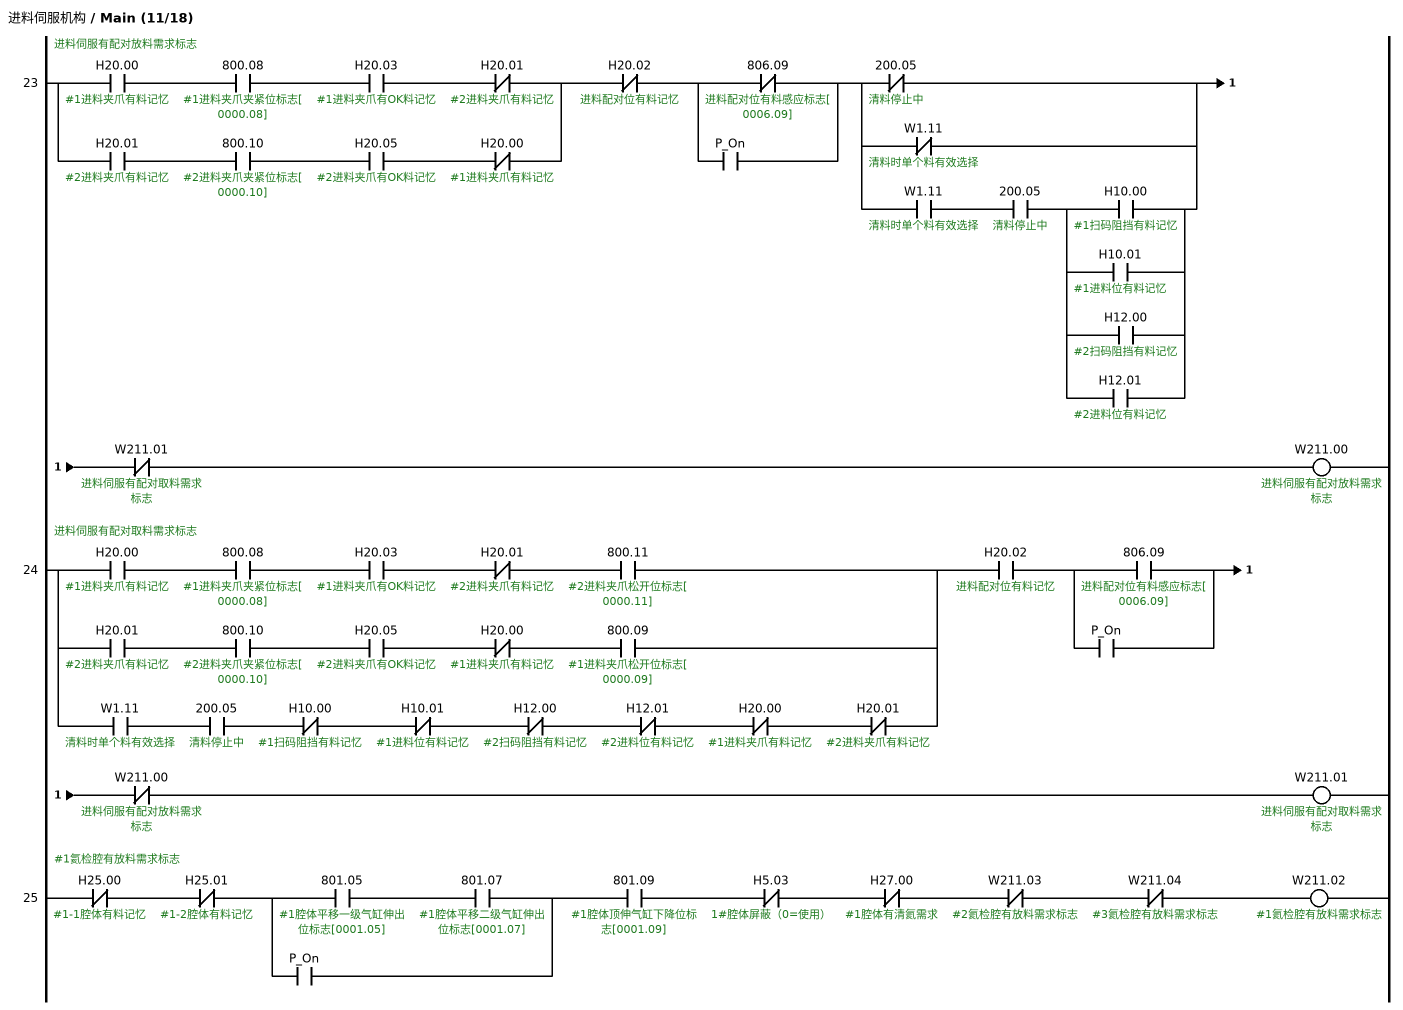
; [picture p72: 进料伺服机构 / Main, rungs 23-25]
; rung 23: 进料伺服有配对放料需求标志
LD H20.00  ; #1进料夹爪有料记忆
AND 800.08  ; #1进料夹爪夹紧位标志[0000.08]
AND H20.03  ; #1进料夹爪有OK料记忆
ANDNOT H20.01  ; #2进料夹爪有料记忆
LD H20.01  ; #2进料夹爪有料记忆
AND 800.10  ; #2进料夹爪夹紧位标志[0000.10]
AND H20.05  ; #2进料夹爪有OK料记忆
ANDNOT H20.00  ; #1进料夹爪有料记忆
ORLD
ANDNOT H20.02  ; 进料配对位有料记忆
LDNOT 806.09  ; 进料配对位有料感应标志[0006.09]
OR P_On
ANDLD
LDNOT 200.05  ; 清料停止中
ORNOT W1.11  ; 清料时单个料有效选择
LD W1.11  ; 清料时单个料有效选择
AND 200.05  ; 清料停止中
LD H10.00  ; #1扫码阻挡有料记忆
OR H10.01  ; #1进料位有料记忆
OR H12.00  ; #2扫码阻挡有料记忆
OR H12.01  ; #2进料位有料记忆
ANDLD
ORLD
ANDLD
ANDNOT W211.01  ; 进料伺服有配对取料需求标志
OUT W211.00  ; 进料伺服有配对放料需求标志
; rung 24: 进料伺服有配对取料需求标志
LD H20.00  ; #1进料夹爪有料记忆
AND 800.08  ; #1进料夹爪夹紧位标志[0000.08]
AND H20.03  ; #1进料夹爪有OK料记忆
ANDNOT H20.01  ; #2进料夹爪有料记忆
AND 800.11  ; #2进料夹爪松开位标志[0000.11]
LD H20.01  ; #2进料夹爪有料记忆
AND 800.10  ; #2进料夹爪夹紧位标志[0000.10]
AND H20.05  ; #2进料夹爪有OK料记忆
ANDNOT H20.00  ; #1进料夹爪有料记忆
AND 800.09  ; #1进料夹爪松开位标志[0000.09]
ORLD
LD W1.11  ; 清料时单个料有效选择
AND 200.05  ; 清料停止中
ANDNOT H10.00  ; #1扫码阻挡有料记忆
ANDNOT H10.01  ; #1进料位有料记忆
ANDNOT H12.00  ; #2扫码阻挡有料记忆
ANDNOT H12.01  ; #2进料位有料记忆
ANDNOT H20.00  ; #1进料夹爪有料记忆
ANDNOT H20.01  ; #2进料夹爪有料记忆
ORLD
AND H20.02  ; 进料配对位有料记忆
LD 806.09  ; 进料配对位有料感应标志[0006.09]
OR P_On
ANDLD
ANDNOT W211.00  ; 进料伺服有配对放料需求标志
OUT W211.01  ; 进料伺服有配对取料需求标志
; rung 25: #1氦检腔有放料需求标志
LDNOT H25.00  ; #1-1腔体有料记忆
ANDNOT H25.01  ; #1-2腔体有料记忆
LD 801.05  ; #1腔体平移一级气缸伸出位标志[0001.05]
AND 801.07  ; #1腔体平移二级气缸伸出位标志[0001.07]
OR P_On
ANDLD
AND 801.09  ; #1腔体顶伸气缸下降位标志[0001.09]
ANDNOT H5.03  ; 1#腔体屏蔽（0=使用）
ANDNOT H27.00  ; #1腔体有清氦需求
ANDNOT W211.03  ; #2氦检腔有放料需求标志
ANDNOT W211.04  ; #3氦检腔有放料需求标志
OUT W211.02  ; #1氦检腔有放料需求标志

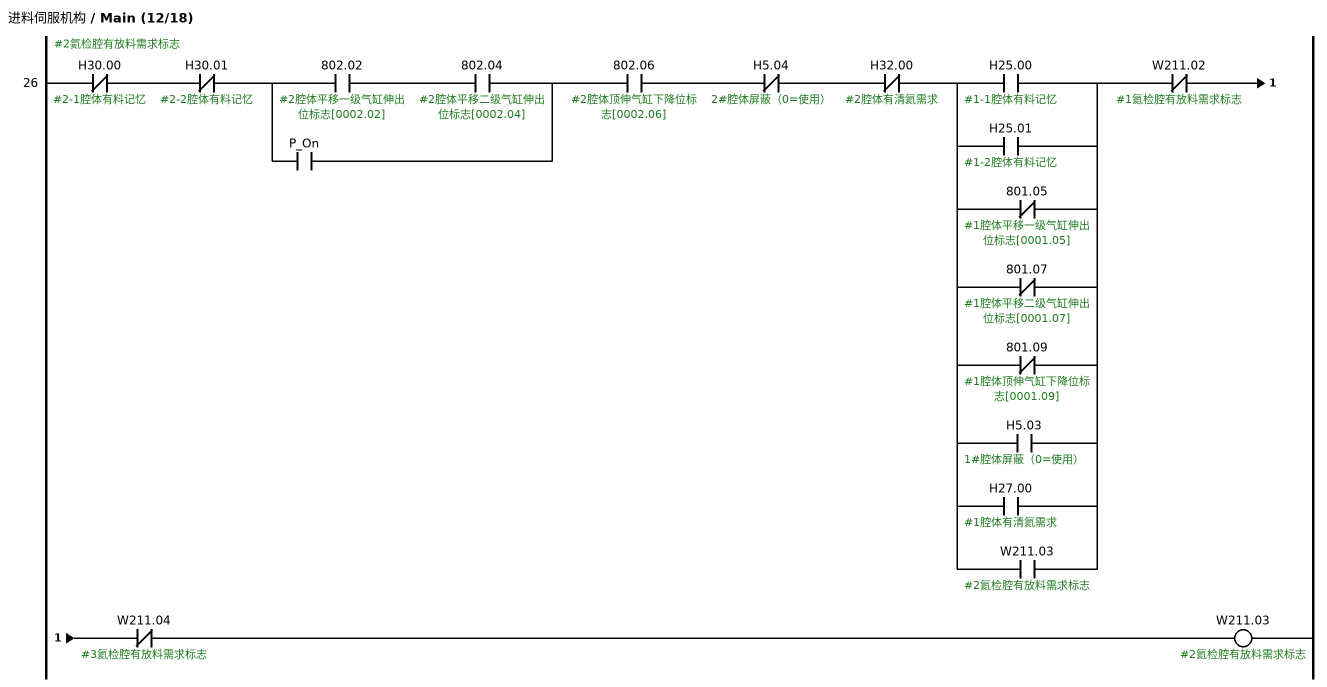
; rung 26: #2氦检腔有放料需求标志
LDNOT H30.00  ; #2-1腔体有料记忆
ANDNOT H30.01  ; #2-2腔体有料记忆
LD 802.02  ; #2腔体平移一级气缸伸出位标志[0002.02]
AND 802.04  ; #2腔体平移二级气缸伸出位标志[0002.04]
OR P_On
ANDLD
AND 802.06  ; #2腔体顶伸气缸下降位标志[0002.06]
ANDNOT H5.04  ; 2#腔体屏蔽（0=使用）
ANDNOT H32.00  ; #2腔体有清氦需求
LD H25.00  ; #1-1腔体有料记忆
OR H25.01  ; #1-2腔体有料记忆
ORNOT 801.05  ; #1腔体平移一级气缸伸出位标志[0001.05]
ORNOT 801.07  ; #1腔体平移二级气缸伸出位标志[0001.07]
ORNOT 801.09  ; #1腔体顶伸气缸下降位标志[0001.09]
OR H5.03  ; 1#腔体屏蔽（0=使用）
OR H27.00  ; #1腔体有清氦需求
OR W211.03  ; #2氦检腔有放料需求标志
ANDLD
ANDNOT W211.02  ; #1氦检腔有放料需求标志
ANDNOT W211.04  ; #3氦检腔有放料需求标志
OUT W211.03  ; #2氦检腔有放料需求标志

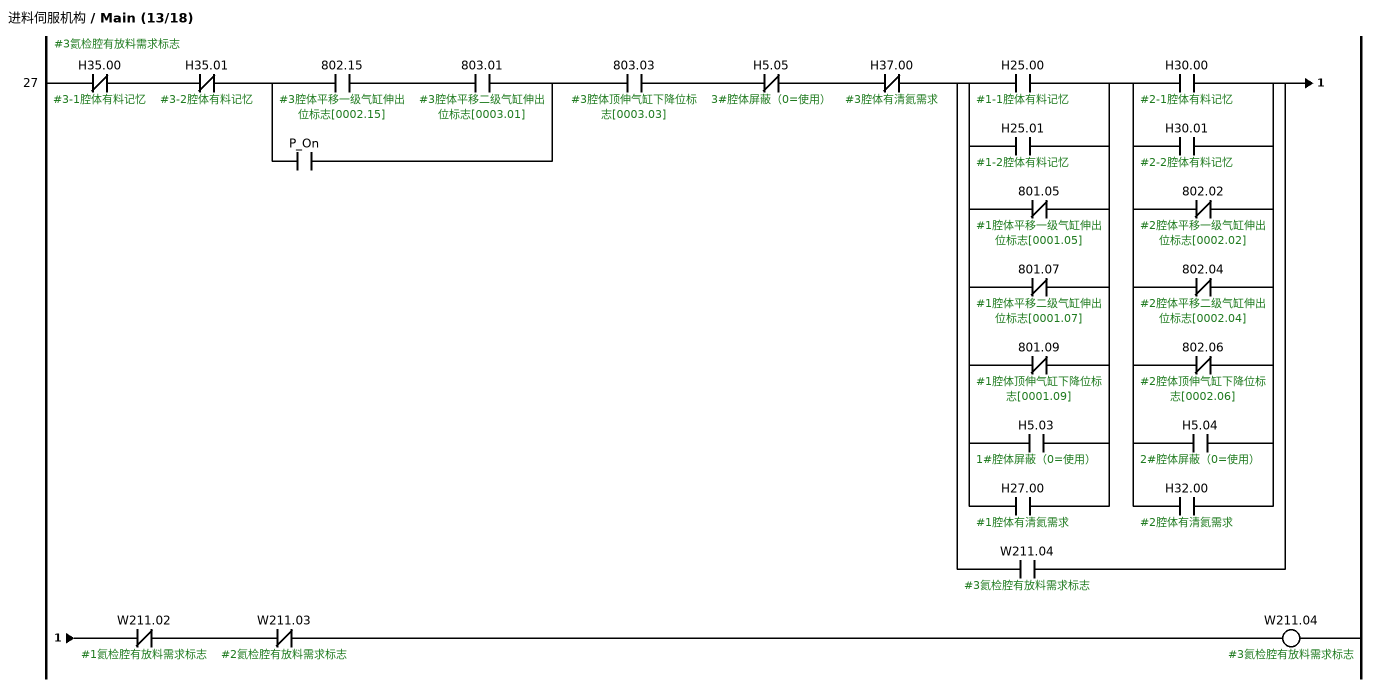
; rung 27: #3氦检腔有放料需求标志
LDNOT H35.00  ; #3-1腔体有料记忆
ANDNOT H35.01  ; #3-2腔体有料记忆
LD 802.15  ; #3腔体平移一级气缸伸出位标志[0002.15]
AND 803.01  ; #3腔体平移二级气缸伸出位标志[0003.01]
OR P_On
ANDLD
AND 803.03  ; #3腔体顶伸气缸下降位标志[0003.03]
ANDNOT H5.05  ; 3#腔体屏蔽（0=使用）
ANDNOT H37.00  ; #3腔体有清氦需求
LD H25.00  ; #1-1腔体有料记忆
OR H25.01  ; #1-2腔体有料记忆
ORNOT 801.05  ; #1腔体平移一级气缸伸出位标志[0001.05]
ORNOT 801.07  ; #1腔体平移二级气缸伸出位标志[0001.07]
ORNOT 801.09  ; #1腔体顶伸气缸下降位标志[0001.09]
OR H5.03  ; 1#腔体屏蔽（0=使用）
OR H27.00  ; #1腔体有清氦需求
LD H30.00  ; #2-1腔体有料记忆
OR H30.01  ; #2-2腔体有料记忆
ORNOT 802.02  ; #2腔体平移一级气缸伸出位标志[0002.02]
ORNOT 802.04  ; #2腔体平移二级气缸伸出位标志[0002.04]
ORNOT 802.06  ; #2腔体顶伸气缸下降位标志[0002.06]
OR H5.04  ; 2#腔体屏蔽（0=使用）
OR H32.00  ; #2腔体有清氦需求
ANDLD
OR W211.04  ; #3氦检腔有放料需求标志
ANDLD
ANDNOT W211.02  ; #1氦检腔有放料需求标志
ANDNOT W211.03  ; #2氦检腔有放料需求标志
OUT W211.04  ; #3氦检腔有放料需求标志

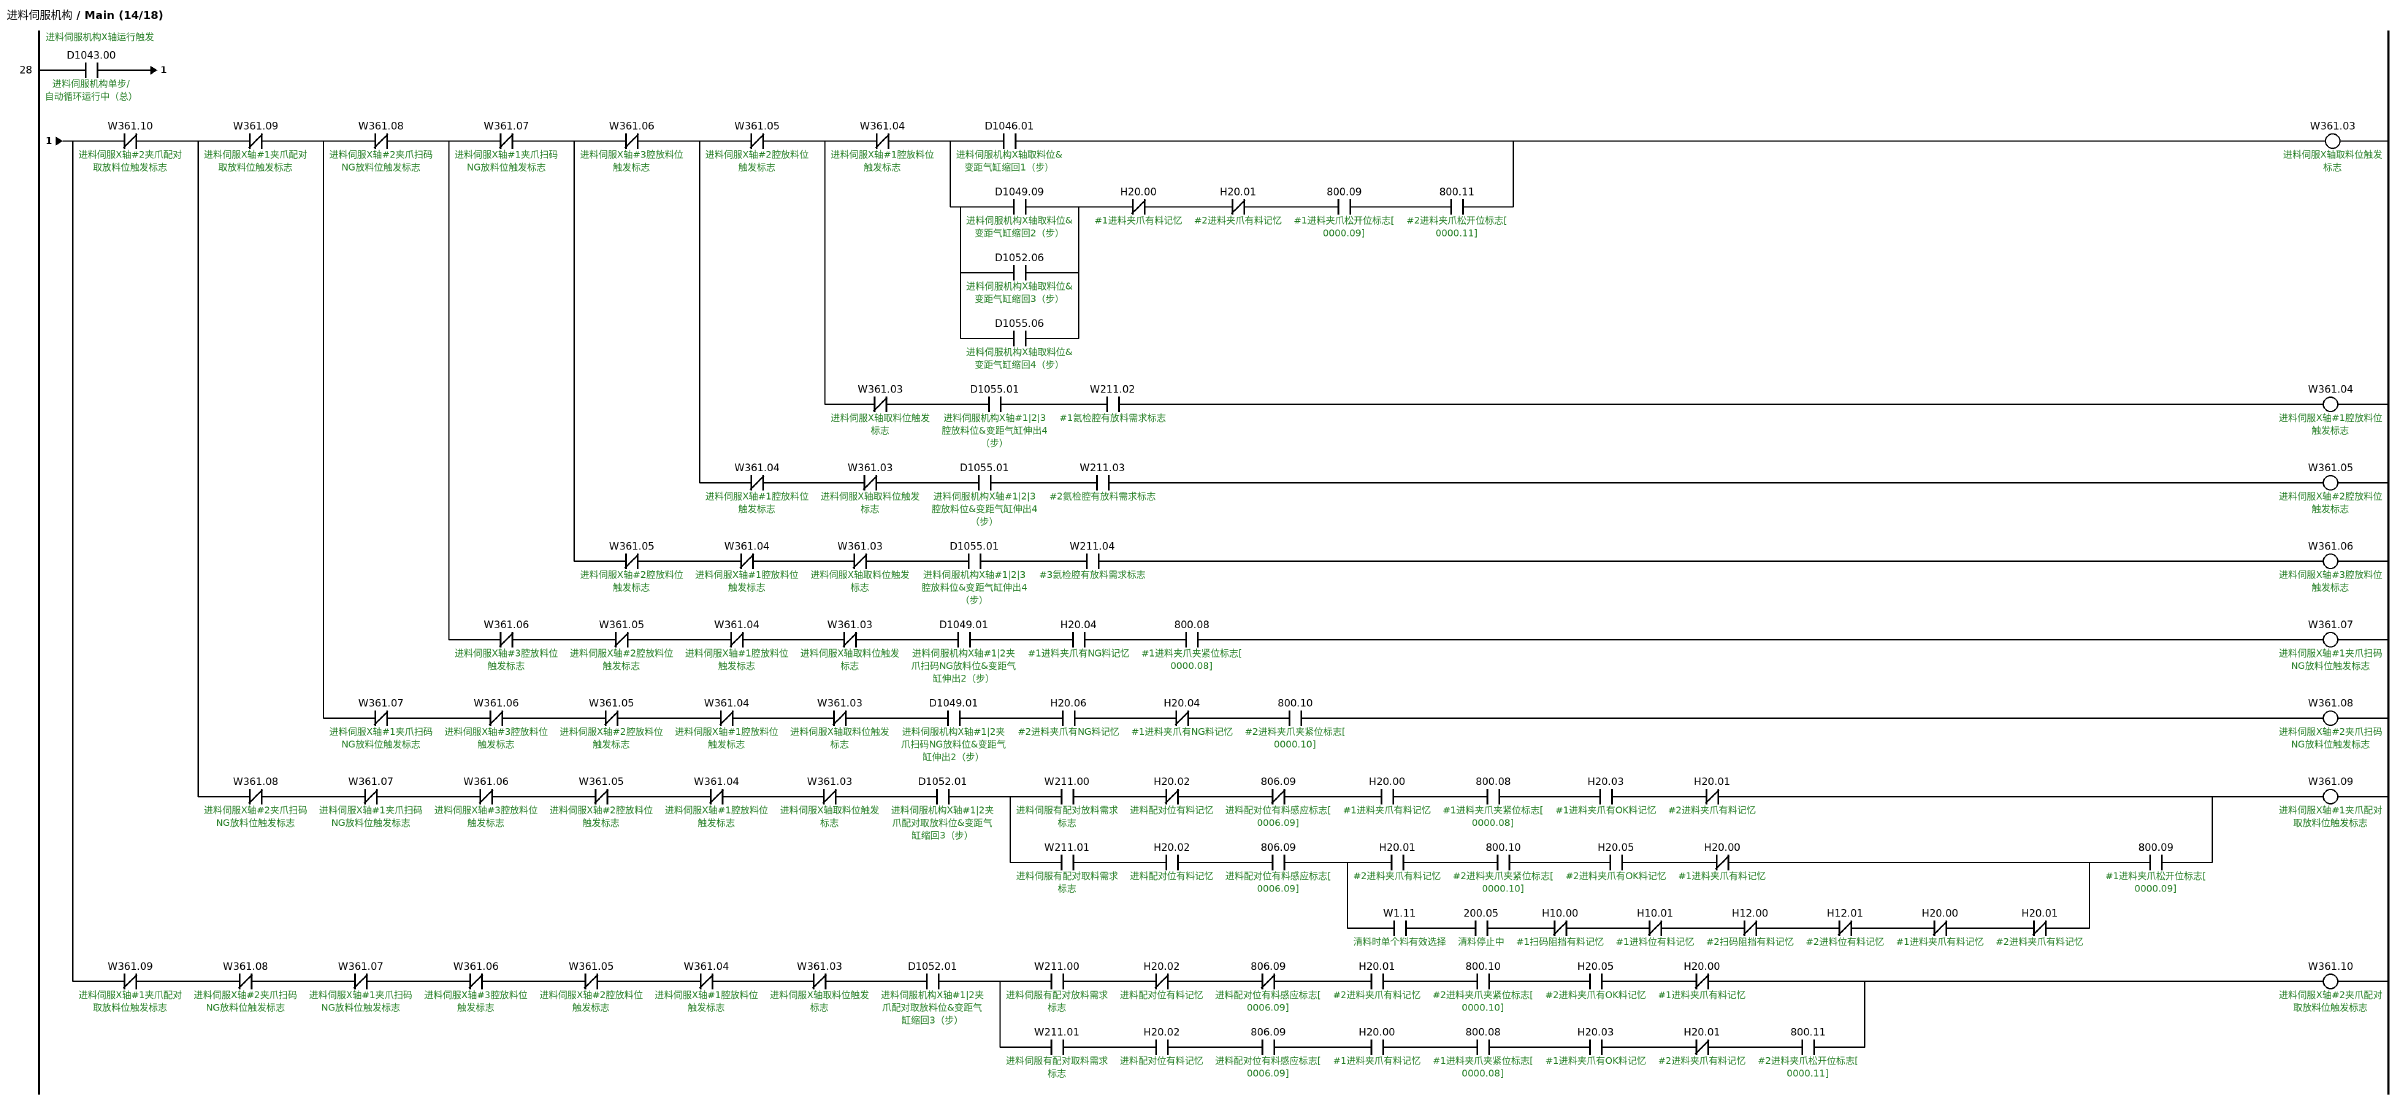
; rung 28: 进料伺服机构X轴运行触发
LD D1043.00  ; 进料伺服机构单步/自动循环运行中（总）
OUT TR0
ANDNOT W361.10  ; 进料伺服X轴#2夹爪配对取放料位触发标志
OUT TR1
ANDNOT W361.09  ; 进料伺服X轴#1夹爪配对取放料位触发标志
OUT TR2
ANDNOT W361.08  ; 进料伺服X轴#2夹爪扫码NG放料位触发标志
OUT TR3
ANDNOT W361.07  ; 进料伺服X轴#1夹爪扫码NG放料位触发标志
OUT TR4
ANDNOT W361.06  ; 进料伺服X轴#3腔放料位触发标志
OUT TR5
ANDNOT W361.05  ; 进料伺服X轴#2腔放料位触发标志
OUT TR6
ANDNOT W361.04  ; 进料伺服X轴#1腔放料位触发标志
LD D1046.01  ; 进料伺服机构X轴取料位&变距气缸缩回1（步）
LD D1049.09  ; 进料伺服机构X轴取料位&变距气缸缩回2（步）
OR D1052.06  ; 进料伺服机构X轴取料位&变距气缸缩回3（步）
OR D1055.06  ; 进料伺服机构X轴取料位&变距气缸缩回4（步）
ANDNOT H20.00  ; #1进料夹爪有料记忆
ANDNOT H20.01  ; #2进料夹爪有料记忆
AND 800.09  ; #1进料夹爪松开位标志[0000.09]
AND 800.11  ; #2进料夹爪松开位标志[0000.11]
ORLD
ANDLD
OUT W361.03  ; 进料伺服X轴取料位触发标志
LD TR6
ANDNOT W361.03  ; 进料伺服X轴取料位触发标志
AND D1055.01  ; 进料伺服机构X轴#1|2|3腔放料位&变距气缸伸出4（步）
AND W211.02  ; #1氦检腔有放料需求标志
OUT W361.04  ; 进料伺服X轴#1腔放料位触发标志
LD TR5
ANDNOT W361.04  ; 进料伺服X轴#1腔放料位触发标志
ANDNOT W361.03  ; 进料伺服X轴取料位触发标志
AND D1055.01  ; 进料伺服机构X轴#1|2|3腔放料位&变距气缸伸出4（步）
AND W211.03  ; #2氦检腔有放料需求标志
OUT W361.05  ; 进料伺服X轴#2腔放料位触发标志
LD TR4
ANDNOT W361.05  ; 进料伺服X轴#2腔放料位触发标志
ANDNOT W361.04  ; 进料伺服X轴#1腔放料位触发标志
ANDNOT W361.03  ; 进料伺服X轴取料位触发标志
AND D1055.01  ; 进料伺服机构X轴#1|2|3腔放料位&变距气缸伸出4（步）
AND W211.04  ; #3氦检腔有放料需求标志
OUT W361.06  ; 进料伺服X轴#3腔放料位触发标志
LD TR3
ANDNOT W361.06  ; 进料伺服X轴#3腔放料位触发标志
ANDNOT W361.05  ; 进料伺服X轴#2腔放料位触发标志
ANDNOT W361.04  ; 进料伺服X轴#1腔放料位触发标志
ANDNOT W361.03  ; 进料伺服X轴取料位触发标志
AND D1049.01  ; 进料伺服机构X轴#1|2夹爪扫码NG放料位&变距气缸伸出2（步）
AND H20.04  ; #1进料夹爪有NG料记忆
AND 800.08  ; #1进料夹爪夹紧位标志[0000.08]
OUT W361.07  ; 进料伺服X轴#1夹爪扫码NG放料位触发标志
LD TR2
ANDNOT W361.07  ; 进料伺服X轴#1夹爪扫码NG放料位触发标志
ANDNOT W361.06  ; 进料伺服X轴#3腔放料位触发标志
ANDNOT W361.05  ; 进料伺服X轴#2腔放料位触发标志
ANDNOT W361.04  ; 进料伺服X轴#1腔放料位触发标志
ANDNOT W361.03  ; 进料伺服X轴取料位触发标志
AND D1049.01  ; 进料伺服机构X轴#1|2夹爪扫码NG放料位&变距气缸伸出2（步）
AND H20.06  ; #2进料夹爪有NG料记忆
ANDNOT H20.04  ; #1进料夹爪有NG料记忆
AND 800.10  ; #2进料夹爪夹紧位标志[0000.10]
OUT W361.08  ; 进料伺服X轴#2夹爪扫码NG放料位触发标志
LD TR1
ANDNOT W361.08  ; 进料伺服X轴#2夹爪扫码NG放料位触发标志
ANDNOT W361.07  ; 进料伺服X轴#1夹爪扫码NG放料位触发标志
ANDNOT W361.06  ; 进料伺服X轴#3腔放料位触发标志
ANDNOT W361.05  ; 进料伺服X轴#2腔放料位触发标志
ANDNOT W361.04  ; 进料伺服X轴#1腔放料位触发标志
ANDNOT W361.03  ; 进料伺服X轴取料位触发标志
AND D1052.01  ; 进料伺服机构X轴#1|2夹爪配对取放料位&变距气缸缩回3（步）
LD W211.00  ; 进料伺服有配对放料需求标志
ANDNOT H20.02  ; 进料配对位有料记忆
ANDNOT 806.09  ; 进料配对位有料感应标志[0006.09]
AND H20.00  ; #1进料夹爪有料记忆
AND 800.08  ; #1进料夹爪夹紧位标志[0000.08]
AND H20.03  ; #1进料夹爪有OK料记忆
ANDNOT H20.01  ; #2进料夹爪有料记忆
LD W211.01  ; 进料伺服有配对取料需求标志
AND H20.02  ; 进料配对位有料记忆
AND 806.09  ; 进料配对位有料感应标志[0006.09]
LD H20.01  ; #2进料夹爪有料记忆
AND 800.10  ; #2进料夹爪夹紧位标志[0000.10]
AND H20.05  ; #2进料夹爪有OK料记忆
ANDNOT H20.00  ; #1进料夹爪有料记忆
LD W1.11  ; 清料时单个料有效选择
AND 200.05  ; 清料停止中
ANDNOT H10.00  ; #1扫码阻挡有料记忆
ANDNOT H10.01  ; #1进料位有料记忆
ANDNOT H12.00  ; #2扫码阻挡有料记忆
ANDNOT H12.01  ; #2进料位有料记忆
ANDNOT H20.00  ; #1进料夹爪有料记忆
ANDNOT H20.01  ; #2进料夹爪有料记忆
ORLD
ANDLD
AND 800.09  ; #1进料夹爪松开位标志[0000.09]
ORLD
ANDLD
OUT W361.09  ; 进料伺服X轴#1夹爪配对取放料位触发标志
LD TR0
ANDNOT W361.09  ; 进料伺服X轴#1夹爪配对取放料位触发标志
ANDNOT W361.08  ; 进料伺服X轴#2夹爪扫码NG放料位触发标志
ANDNOT W361.07  ; 进料伺服X轴#1夹爪扫码NG放料位触发标志
ANDNOT W361.06  ; 进料伺服X轴#3腔放料位触发标志
ANDNOT W361.05  ; 进料伺服X轴#2腔放料位触发标志
ANDNOT W361.04  ; 进料伺服X轴#1腔放料位触发标志
ANDNOT W361.03  ; 进料伺服X轴取料位触发标志
AND D1052.01  ; 进料伺服机构X轴#1|2夹爪配对取放料位&变距气缸缩回3（步）
LD W211.00  ; 进料伺服有配对放料需求标志
ANDNOT H20.02  ; 进料配对位有料记忆
ANDNOT 806.09  ; 进料配对位有料感应标志[0006.09]
AND H20.01  ; #2进料夹爪有料记忆
AND 800.10  ; #2进料夹爪夹紧位标志[0000.10]
AND H20.05  ; #2进料夹爪有OK料记忆
ANDNOT H20.00  ; #1进料夹爪有料记忆
LD W211.01  ; 进料伺服有配对取料需求标志
AND H20.02  ; 进料配对位有料记忆
AND 806.09  ; 进料配对位有料感应标志[0006.09]
AND H20.00  ; #1进料夹爪有料记忆
AND 800.08  ; #1进料夹爪夹紧位标志[0000.08]
AND H20.03  ; #1进料夹爪有OK料记忆
ANDNOT H20.01  ; #2进料夹爪有料记忆
AND 800.11  ; #2进料夹爪松开位标志[0000.11]
ORLD
ANDLD
OUT W361.10  ; 进料伺服X轴#2夹爪配对取放料位触发标志

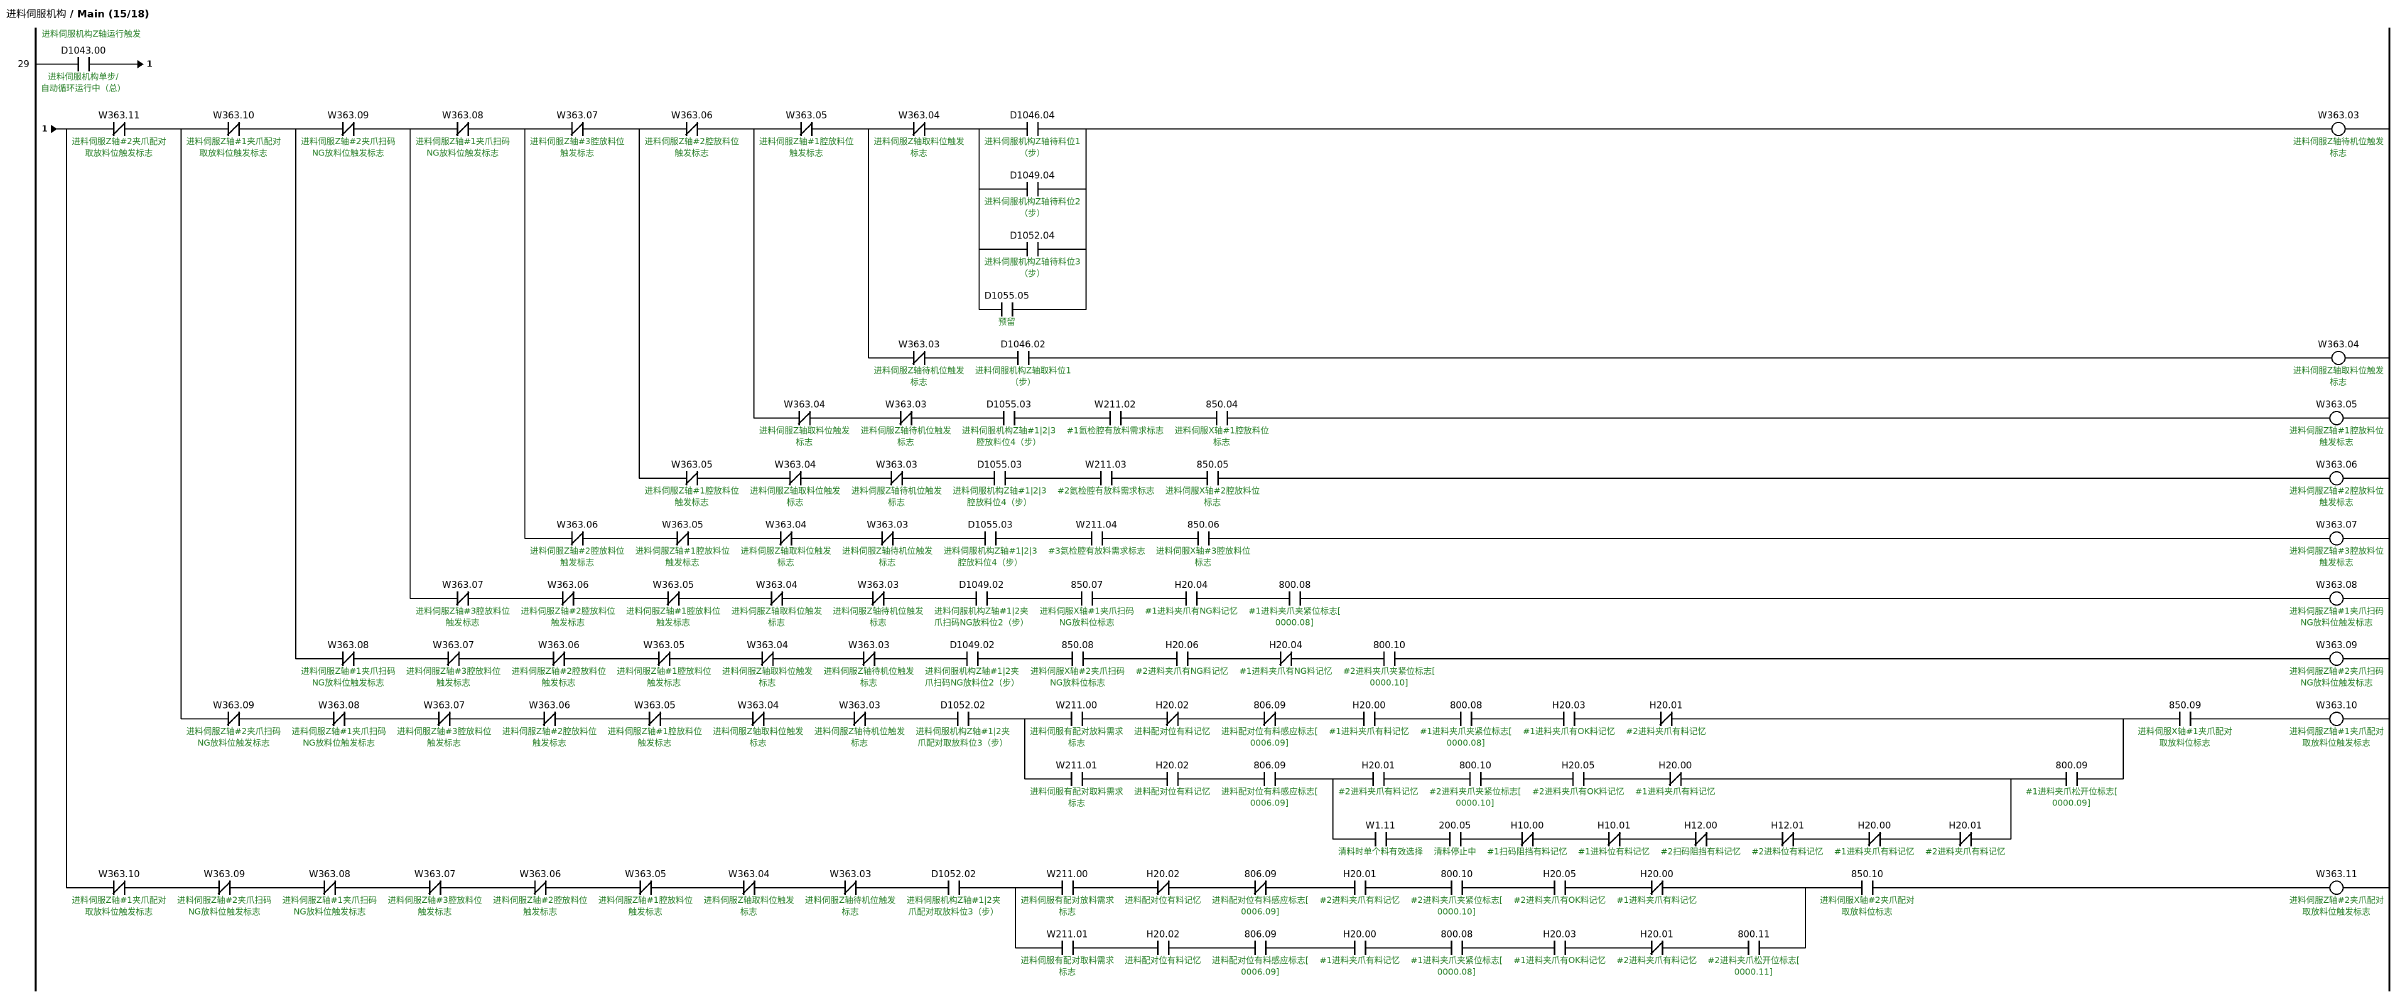
; rung 29: 进料伺服机构Z轴运行触发
LD D1043.00  ; 进料伺服机构单步/自动循环运行中（总）
OUT TR0
ANDNOT W363.11  ; 进料伺服Z轴#2夹爪配对取放料位触发标志
OUT TR1
ANDNOT W363.10  ; 进料伺服Z轴#1夹爪配对取放料位触发标志
OUT TR2
ANDNOT W363.09  ; 进料伺服Z轴#2夹爪扫码NG放料位触发标志
OUT TR3
ANDNOT W363.08  ; 进料伺服Z轴#1夹爪扫码NG放料位触发标志
OUT TR4
ANDNOT W363.07  ; 进料伺服Z轴#3腔放料位触发标志
OUT TR5
ANDNOT W363.06  ; 进料伺服Z轴#2腔放料位触发标志
OUT TR6
ANDNOT W363.05  ; 进料伺服Z轴#1腔放料位触发标志
OUT TR7
ANDNOT W363.04  ; 进料伺服Z轴取料位触发标志
LD D1046.04  ; 进料伺服机构Z轴待料位1（步）
OR D1049.04  ; 进料伺服机构Z轴待料位2（步）
OR D1052.04  ; 进料伺服机构Z轴待料位3（步）
OR D1055.05  ; 预留
ANDLD
OUT W363.03  ; 进料伺服Z轴待机位触发标志
LD TR7
ANDNOT W363.03  ; 进料伺服Z轴待机位触发标志
AND D1046.02  ; 进料伺服机构Z轴取料位1（步）
OUT W363.04  ; 进料伺服Z轴取料位触发标志
LD TR6
ANDNOT W363.04  ; 进料伺服Z轴取料位触发标志
ANDNOT W363.03  ; 进料伺服Z轴待机位触发标志
AND D1055.03  ; 进料伺服机构Z轴#1|2|3腔放料位4（步）
AND W211.02  ; #1氦检腔有放料需求标志
AND 850.04  ; 进料伺服X轴#1腔放料位标志
OUT W363.05  ; 进料伺服Z轴#1腔放料位触发标志
LD TR5
ANDNOT W363.05  ; 进料伺服Z轴#1腔放料位触发标志
ANDNOT W363.04  ; 进料伺服Z轴取料位触发标志
ANDNOT W363.03  ; 进料伺服Z轴待机位触发标志
AND D1055.03  ; 进料伺服机构Z轴#1|2|3腔放料位4（步）
AND W211.03  ; #2氦检腔有放料需求标志
AND 850.05  ; 进料伺服X轴#2腔放料位标志
OUT W363.06  ; 进料伺服Z轴#2腔放料位触发标志
LD TR4
ANDNOT W363.06  ; 进料伺服Z轴#2腔放料位触发标志
ANDNOT W363.05  ; 进料伺服Z轴#1腔放料位触发标志
ANDNOT W363.04  ; 进料伺服Z轴取料位触发标志
ANDNOT W363.03  ; 进料伺服Z轴待机位触发标志
AND D1055.03  ; 进料伺服机构Z轴#1|2|3腔放料位4（步）
AND W211.04  ; #3氦检腔有放料需求标志
AND 850.06  ; 进料伺服X轴#3腔放料位标志
OUT W363.07  ; 进料伺服Z轴#3腔放料位触发标志
LD TR3
ANDNOT W363.07  ; 进料伺服Z轴#3腔放料位触发标志
ANDNOT W363.06  ; 进料伺服Z轴#2腔放料位触发标志
ANDNOT W363.05  ; 进料伺服Z轴#1腔放料位触发标志
ANDNOT W363.04  ; 进料伺服Z轴取料位触发标志
ANDNOT W363.03  ; 进料伺服Z轴待机位触发标志
AND D1049.02  ; 进料伺服机构Z轴#1|2夹爪扫码NG放料位2（步）
AND 850.07  ; 进料伺服X轴#1夹爪扫码NG放料位标志
AND H20.04  ; #1进料夹爪有NG料记忆
AND 800.08  ; #1进料夹爪夹紧位标志[0000.08]
OUT W363.08  ; 进料伺服Z轴#1夹爪扫码NG放料位触发标志
LD TR2
ANDNOT W363.08  ; 进料伺服Z轴#1夹爪扫码NG放料位触发标志
ANDNOT W363.07  ; 进料伺服Z轴#3腔放料位触发标志
ANDNOT W363.06  ; 进料伺服Z轴#2腔放料位触发标志
ANDNOT W363.05  ; 进料伺服Z轴#1腔放料位触发标志
ANDNOT W363.04  ; 进料伺服Z轴取料位触发标志
ANDNOT W363.03  ; 进料伺服Z轴待机位触发标志
AND D1049.02  ; 进料伺服机构Z轴#1|2夹爪扫码NG放料位2（步）
AND 850.08  ; 进料伺服X轴#2夹爪扫码NG放料位标志
AND H20.06  ; #2进料夹爪有NG料记忆
ANDNOT H20.04  ; #1进料夹爪有NG料记忆
AND 800.10  ; #2进料夹爪夹紧位标志[0000.10]
OUT W363.09  ; 进料伺服Z轴#2夹爪扫码NG放料位触发标志
LD TR1
ANDNOT W363.09  ; 进料伺服Z轴#2夹爪扫码NG放料位触发标志
ANDNOT W363.08  ; 进料伺服Z轴#1夹爪扫码NG放料位触发标志
ANDNOT W363.07  ; 进料伺服Z轴#3腔放料位触发标志
ANDNOT W363.06  ; 进料伺服Z轴#2腔放料位触发标志
ANDNOT W363.05  ; 进料伺服Z轴#1腔放料位触发标志
ANDNOT W363.04  ; 进料伺服Z轴取料位触发标志
ANDNOT W363.03  ; 进料伺服Z轴待机位触发标志
AND D1052.02  ; 进料伺服机构Z轴#1|2夹爪配对取放料位3（步）
LD W211.00  ; 进料伺服有配对放料需求标志
ANDNOT H20.02  ; 进料配对位有料记忆
ANDNOT 806.09  ; 进料配对位有料感应标志[0006.09]
AND H20.00  ; #1进料夹爪有料记忆
AND 800.08  ; #1进料夹爪夹紧位标志[0000.08]
AND H20.03  ; #1进料夹爪有OK料记忆
ANDNOT H20.01  ; #2进料夹爪有料记忆
LD W211.01  ; 进料伺服有配对取料需求标志
AND H20.02  ; 进料配对位有料记忆
AND 806.09  ; 进料配对位有料感应标志[0006.09]
LD H20.01  ; #2进料夹爪有料记忆
AND 800.10  ; #2进料夹爪夹紧位标志[0000.10]
AND H20.05  ; #2进料夹爪有OK料记忆
ANDNOT H20.00  ; #1进料夹爪有料记忆
LD W1.11  ; 清料时单个料有效选择
AND 200.05  ; 清料停止中
ANDNOT H10.00  ; #1扫码阻挡有料记忆
ANDNOT H10.01  ; #1进料位有料记忆
ANDNOT H12.00  ; #2扫码阻挡有料记忆
ANDNOT H12.01  ; #2进料位有料记忆
ANDNOT H20.00  ; #1进料夹爪有料记忆
ANDNOT H20.01  ; #2进料夹爪有料记忆
ORLD
ANDLD
AND 800.09  ; #1进料夹爪松开位标志[0000.09]
ORLD
ANDLD
AND 850.09  ; 进料伺服X轴#1夹爪配对取放料位标志
OUT W363.10  ; 进料伺服Z轴#1夹爪配对取放料位触发标志
LD TR0
ANDNOT W363.10  ; 进料伺服Z轴#1夹爪配对取放料位触发标志
ANDNOT W363.09  ; 进料伺服Z轴#2夹爪扫码NG放料位触发标志
ANDNOT W363.08  ; 进料伺服Z轴#1夹爪扫码NG放料位触发标志
ANDNOT W363.07  ; 进料伺服Z轴#3腔放料位触发标志
ANDNOT W363.06  ; 进料伺服Z轴#2腔放料位触发标志
ANDNOT W363.05  ; 进料伺服Z轴#1腔放料位触发标志
ANDNOT W363.04  ; 进料伺服Z轴取料位触发标志
ANDNOT W363.03  ; 进料伺服Z轴待机位触发标志
AND D1052.02  ; 进料伺服机构Z轴#1|2夹爪配对取放料位3（步）
LD W211.00  ; 进料伺服有配对放料需求标志
ANDNOT H20.02  ; 进料配对位有料记忆
ANDNOT 806.09  ; 进料配对位有料感应标志[0006.09]
AND H20.01  ; #2进料夹爪有料记忆
AND 800.10  ; #2进料夹爪夹紧位标志[0000.10]
AND H20.05  ; #2进料夹爪有OK料记忆
ANDNOT H20.00  ; #1进料夹爪有料记忆
LD W211.01  ; 进料伺服有配对取料需求标志
AND H20.02  ; 进料配对位有料记忆
AND 806.09  ; 进料配对位有料感应标志[0006.09]
AND H20.00  ; #1进料夹爪有料记忆
AND 800.08  ; #1进料夹爪夹紧位标志[0000.08]
AND H20.03  ; #1进料夹爪有OK料记忆
ANDNOT H20.01  ; #2进料夹爪有料记忆
AND 800.11  ; #2进料夹爪松开位标志[0000.11]
ORLD
ANDLD
AND 850.10  ; 进料伺服X轴#2夹爪配对取放料位标志
OUT W363.11  ; 进料伺服Z轴#2夹爪配对取放料位触发标志

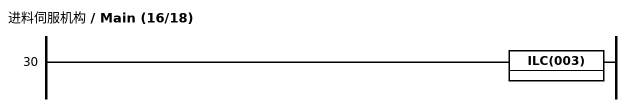
; rung 30
ILC(003)

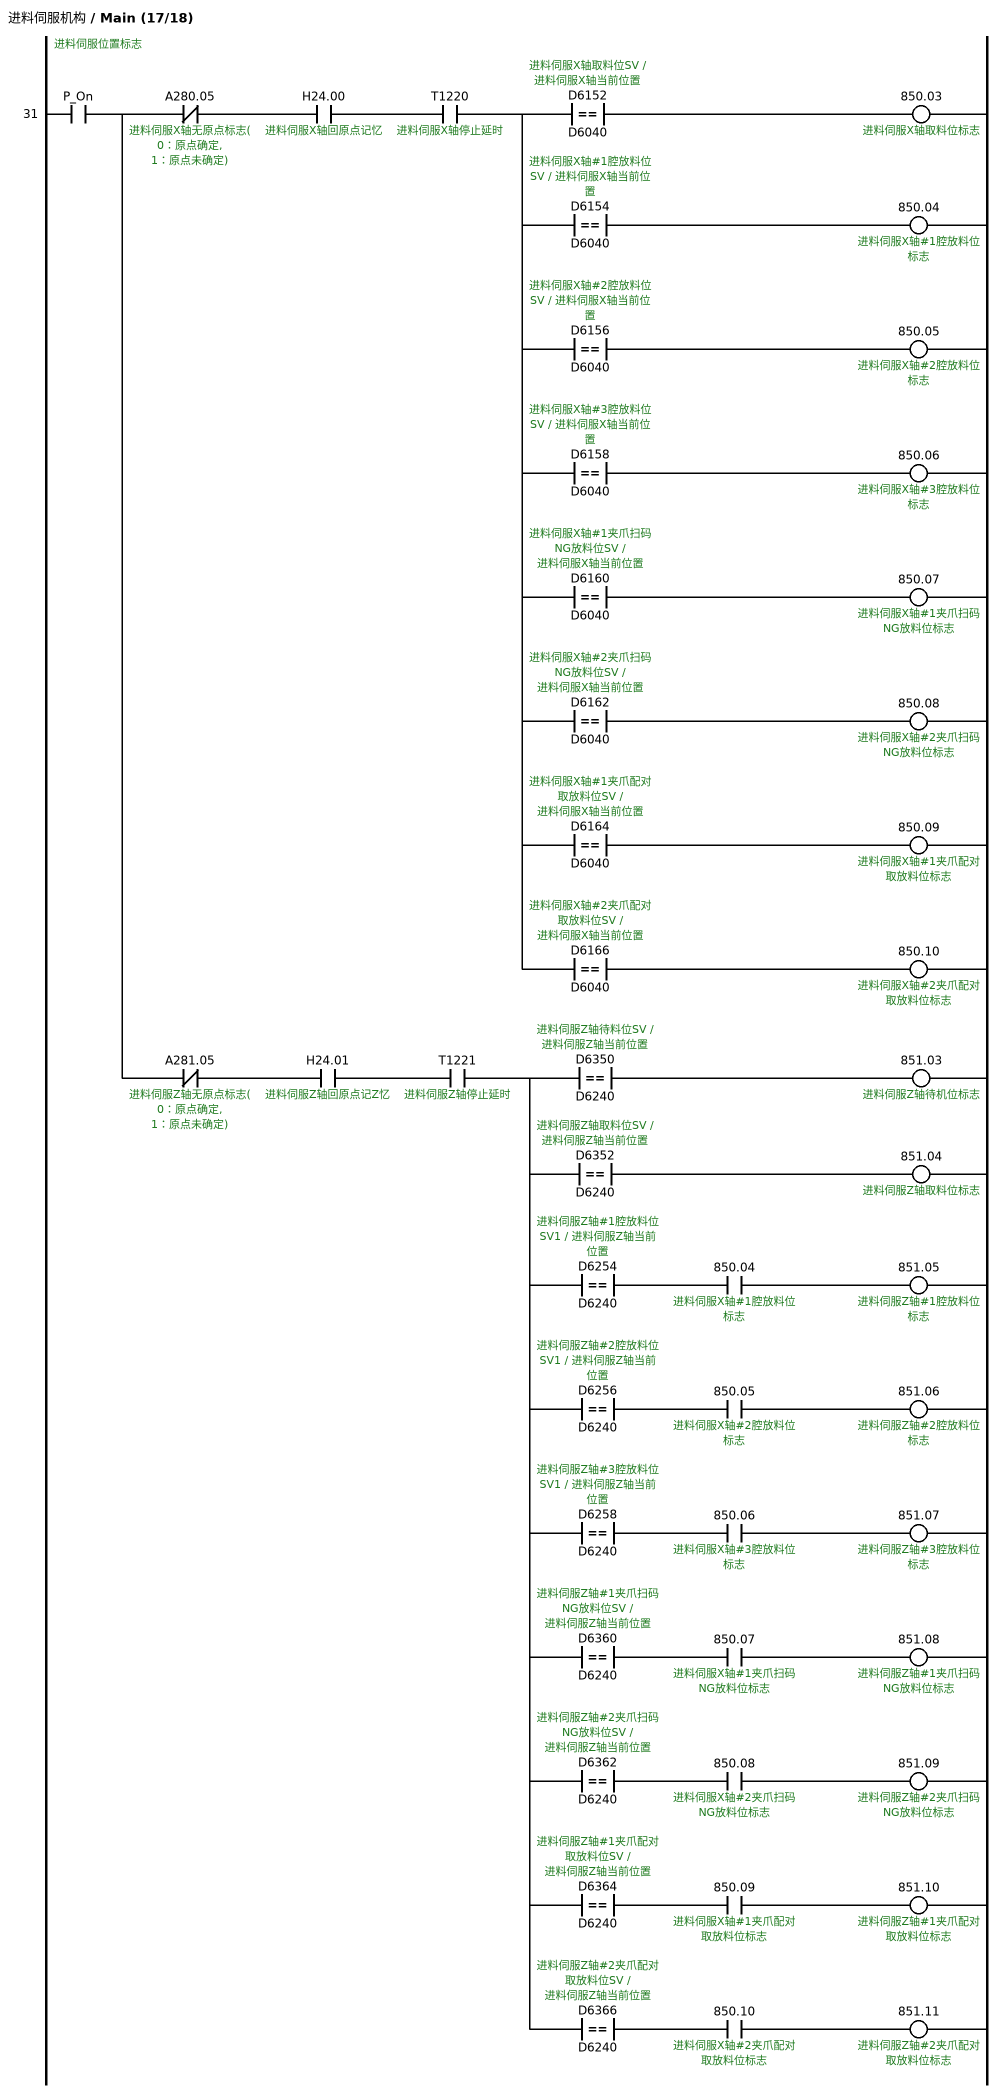
; rung 31: 进料伺服位置标志
LD P_On
OUT TR0
ANDNOT A280.05  ; 进料伺服X轴无原点标志(0：原点确定,1：原点未确定)
AND H24.00  ; 进料伺服X轴回原点记忆
AND T1220  ; 进料伺服X轴停止延时
OUT TR1
AND=SL(303) D6152 D6040  ; 进料伺服X轴取料位SV, 进料伺服X轴当前位置
OUT 850.03  ; 进料伺服X轴取料位标志
LD TR1
AND=SL(303) D6154 D6040  ; 进料伺服X轴#1腔放料位SV, 进料伺服X轴当前位置
OUT 850.04  ; 进料伺服X轴#1腔放料位标志
LD TR1
AND=SL(303) D6156 D6040  ; 进料伺服X轴#2腔放料位SV, 进料伺服X轴当前位置
OUT 850.05  ; 进料伺服X轴#2腔放料位标志
LD TR1
AND=SL(303) D6158 D6040  ; 进料伺服X轴#3腔放料位SV, 进料伺服X轴当前位置
OUT 850.06  ; 进料伺服X轴#3腔放料位标志
LD TR1
AND=SL(303) D6160 D6040  ; 进料伺服X轴#1夹爪扫码NG放料位SV, 进料伺服X轴当前位置
OUT 850.07  ; 进料伺服X轴#1夹爪扫码NG放料位标志
LD TR1
AND=SL(303) D6162 D6040  ; 进料伺服X轴#2夹爪扫码NG放料位SV, 进料伺服X轴当前位置
OUT 850.08  ; 进料伺服X轴#2夹爪扫码NG放料位标志
LD TR1
AND=SL(303) D6164 D6040  ; 进料伺服X轴#1夹爪配对取放料位SV, 进料伺服X轴当前位置
OUT 850.09  ; 进料伺服X轴#1夹爪配对取放料位标志
LD TR1
AND=SL(303) D6166 D6040  ; 进料伺服X轴#2夹爪配对取放料位SV, 进料伺服X轴当前位置
OUT 850.10  ; 进料伺服X轴#2夹爪配对取放料位标志
LD TR0
ANDNOT A281.05  ; 进料伺服Z轴无原点标志(0：原点确定,1：原点未确定)
AND H24.01  ; 进料伺服Z轴回原点记Z忆
AND T1221  ; 进料伺服Z轴停止延时
OUT TR0
AND=SL(303) D6350 D6240  ; 进料伺服Z轴待料位SV, 进料伺服Z轴当前位置
OUT 851.03  ; 进料伺服Z轴待机位标志
LD TR0
AND=SL(303) D6352 D6240  ; 进料伺服Z轴取料位SV, 进料伺服Z轴当前位置
OUT 851.04  ; 进料伺服Z轴取料位标志
LD TR0
AND=SL(303) D6254 D6240  ; 进料伺服Z轴#1腔放料位SV1, 进料伺服Z轴当前位置
AND 850.04  ; 进料伺服X轴#1腔放料位标志
OUT 851.05  ; 进料伺服Z轴#1腔放料位标志
LD TR0
AND=SL(303) D6256 D6240  ; 进料伺服Z轴#2腔放料位SV1, 进料伺服Z轴当前位置
AND 850.05  ; 进料伺服X轴#2腔放料位标志
OUT 851.06  ; 进料伺服Z轴#2腔放料位标志
LD TR0
AND=SL(303) D6258 D6240  ; 进料伺服Z轴#3腔放料位SV1, 进料伺服Z轴当前位置
AND 850.06  ; 进料伺服X轴#3腔放料位标志
OUT 851.07  ; 进料伺服Z轴#3腔放料位标志
LD TR0
AND=SL(303) D6360 D6240  ; 进料伺服Z轴#1夹爪扫码NG放料位SV, 进料伺服Z轴当前位置
AND 850.07  ; 进料伺服X轴#1夹爪扫码NG放料位标志
OUT 851.08  ; 进料伺服Z轴#1夹爪扫码NG放料位标志
LD TR0
AND=SL(303) D6362 D6240  ; 进料伺服Z轴#2夹爪扫码NG放料位SV, 进料伺服Z轴当前位置
AND 850.08  ; 进料伺服X轴#2夹爪扫码NG放料位标志
OUT 851.09  ; 进料伺服Z轴#2夹爪扫码NG放料位标志
LD TR0
AND=SL(303) D6364 D6240  ; 进料伺服Z轴#1夹爪配对取放料位SV, 进料伺服Z轴当前位置
AND 850.09  ; 进料伺服X轴#1夹爪配对取放料位标志
OUT 851.10  ; 进料伺服Z轴#1夹爪配对取放料位标志
LD TR0
AND=SL(303) D6366 D6240  ; 进料伺服Z轴#2夹爪配对取放料位SV, 进料伺服Z轴当前位置
AND 850.10  ; 进料伺服X轴#2夹爪配对取放料位标志
OUT 851.11  ; 进料伺服Z轴#2夹爪配对取放料位标志

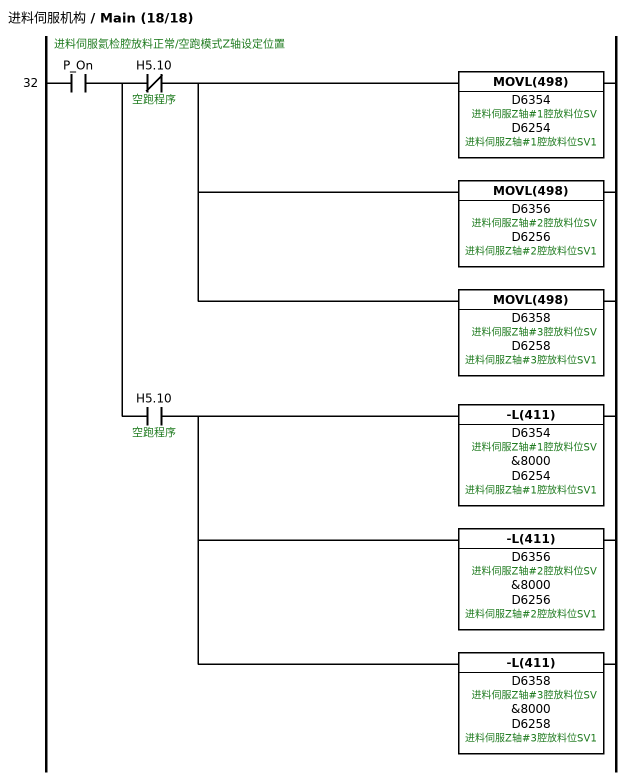
; rung 32: 进料伺服氦检腔放料正常/空跑模式Z轴设定位置
LD P_On
OUT TR0
ANDNOT H5.10  ; 空跑程序
MOVL(498) D6354 D6254  ; 进料伺服Z轴#1腔放料位SV, 进料伺服Z轴#1腔放料位SV1
MOVL(498) D6356 D6256  ; 进料伺服Z轴#2腔放料位SV, 进料伺服Z轴#2腔放料位SV1
MOVL(498) D6358 D6258  ; 进料伺服Z轴#3腔放料位SV, 进料伺服Z轴#3腔放料位SV1
LD TR0
AND H5.10  ; 空跑程序
-L(411) D6354 &8000 D6254  ; 进料伺服Z轴#1腔放料位SV, 进料伺服Z轴#1腔放料位SV1
-L(411) D6356 &8000 D6256  ; 进料伺服Z轴#2腔放料位SV, 进料伺服Z轴#2腔放料位SV1
-L(411) D6358 &8000 D6258  ; 进料伺服Z轴#3腔放料位SV, 进料伺服Z轴#3腔放料位SV1

### Section 进料伺服手动

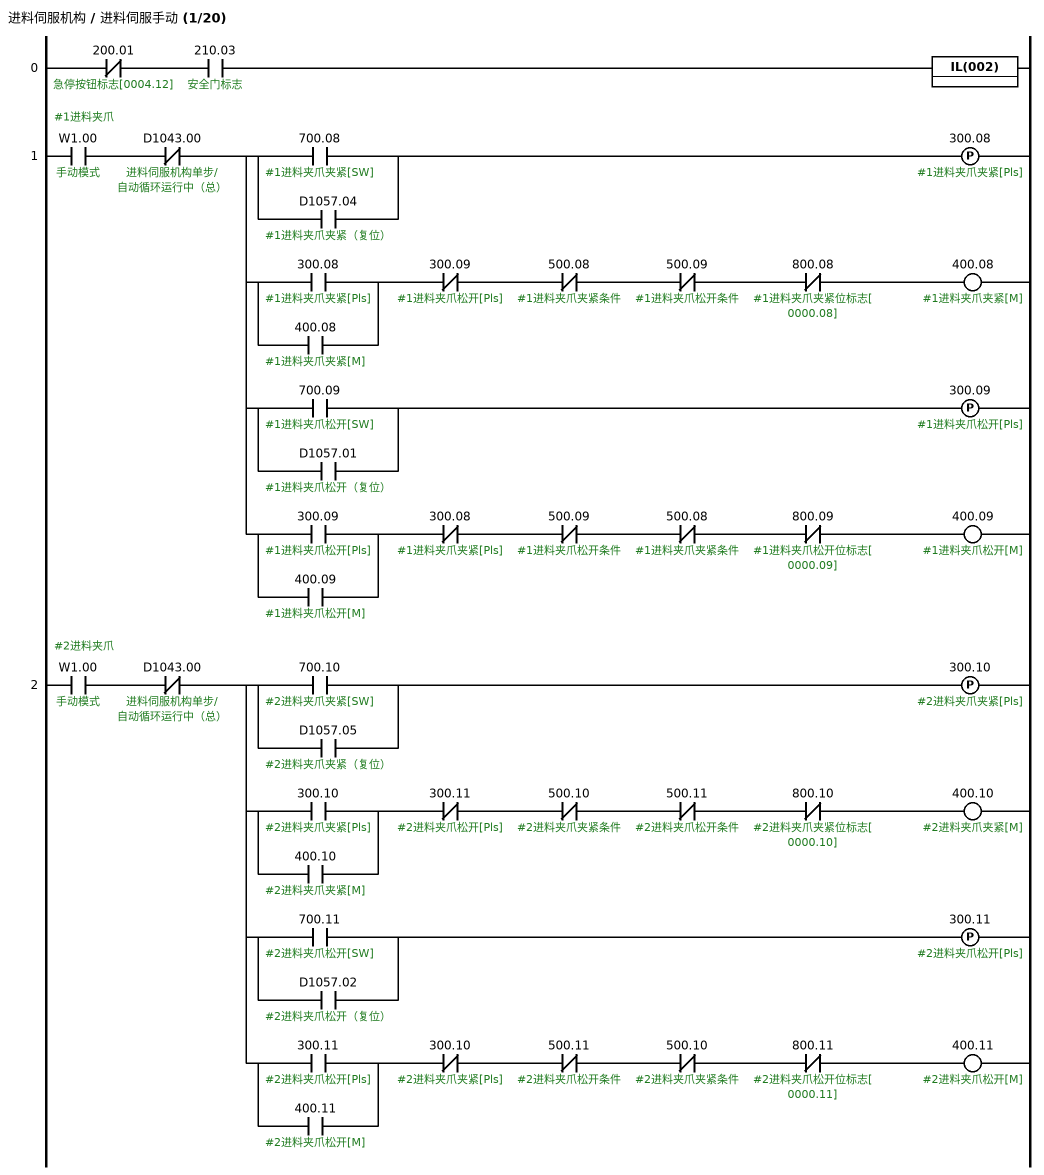
; rung 0
LDNOT 200.01  ; 急停按钮标志[0004.12]
AND 210.03  ; 安全门标志
IL(002)
; rung 1: #1进料夹爪
LD W1.00  ; 手动模式
ANDNOT D1043.00  ; 进料伺服机构单步/自动循环运行中（总）
OUT TR0
LD 700.08  ; #1进料夹爪夹紧[SW]
OR D1057.04  ; #1进料夹爪夹紧（复位）
ANDLD
DIFU(013) 300.08  ; #1进料夹爪夹紧[Pls]
LD TR0
LD 300.08  ; #1进料夹爪夹紧[Pls]
OR 400.08  ; #1进料夹爪夹紧[M]
ANDLD
ANDNOT 300.09  ; #1进料夹爪松开[Pls]
ANDNOT 500.08  ; #1进料夹爪夹紧条件
ANDNOT 500.09  ; #1进料夹爪松开条件
ANDNOT 800.08  ; #1进料夹爪夹紧位标志[0000.08]
OUT 400.08  ; #1进料夹爪夹紧[M]
LD TR0
LD 700.09  ; #1进料夹爪松开[SW]
OR D1057.01  ; #1进料夹爪松开（复位）
ANDLD
DIFU(013) 300.09  ; #1进料夹爪松开[Pls]
LD TR0
LD 300.09  ; #1进料夹爪松开[Pls]
OR 400.09  ; #1进料夹爪松开[M]
ANDLD
ANDNOT 300.08  ; #1进料夹爪夹紧[Pls]
ANDNOT 500.09  ; #1进料夹爪松开条件
ANDNOT 500.08  ; #1进料夹爪夹紧条件
ANDNOT 800.09  ; #1进料夹爪松开位标志[0000.09]
OUT 400.09  ; #1进料夹爪松开[M]
; rung 2: #2进料夹爪
LD W1.00  ; 手动模式
ANDNOT D1043.00  ; 进料伺服机构单步/自动循环运行中（总）
OUT TR0
LD 700.10  ; #2进料夹爪夹紧[SW]
OR D1057.05  ; #2进料夹爪夹紧（复位）
ANDLD
DIFU(013) 300.10  ; #2进料夹爪夹紧[Pls]
LD TR0
LD 300.10  ; #2进料夹爪夹紧[Pls]
OR 400.10  ; #2进料夹爪夹紧[M]
ANDLD
ANDNOT 300.11  ; #2进料夹爪松开[Pls]
ANDNOT 500.10  ; #2进料夹爪夹紧条件
ANDNOT 500.11  ; #2进料夹爪松开条件
ANDNOT 800.10  ; #2进料夹爪夹紧位标志[0000.10]
OUT 400.10  ; #2进料夹爪夹紧[M]
LD TR0
LD 700.11  ; #2进料夹爪松开[SW]
OR D1057.02  ; #2进料夹爪松开（复位）
ANDLD
DIFU(013) 300.11  ; #2进料夹爪松开[Pls]
LD TR0
LD 300.11  ; #2进料夹爪松开[Pls]
OR 400.11  ; #2进料夹爪松开[M]
ANDLD
ANDNOT 300.10  ; #2进料夹爪夹紧[Pls]
ANDNOT 500.11  ; #2进料夹爪松开条件
ANDNOT 500.10  ; #2进料夹爪夹紧条件
ANDNOT 800.11  ; #2进料夹爪松开位标志[0000.11]
OUT 400.11  ; #2进料夹爪松开[M]

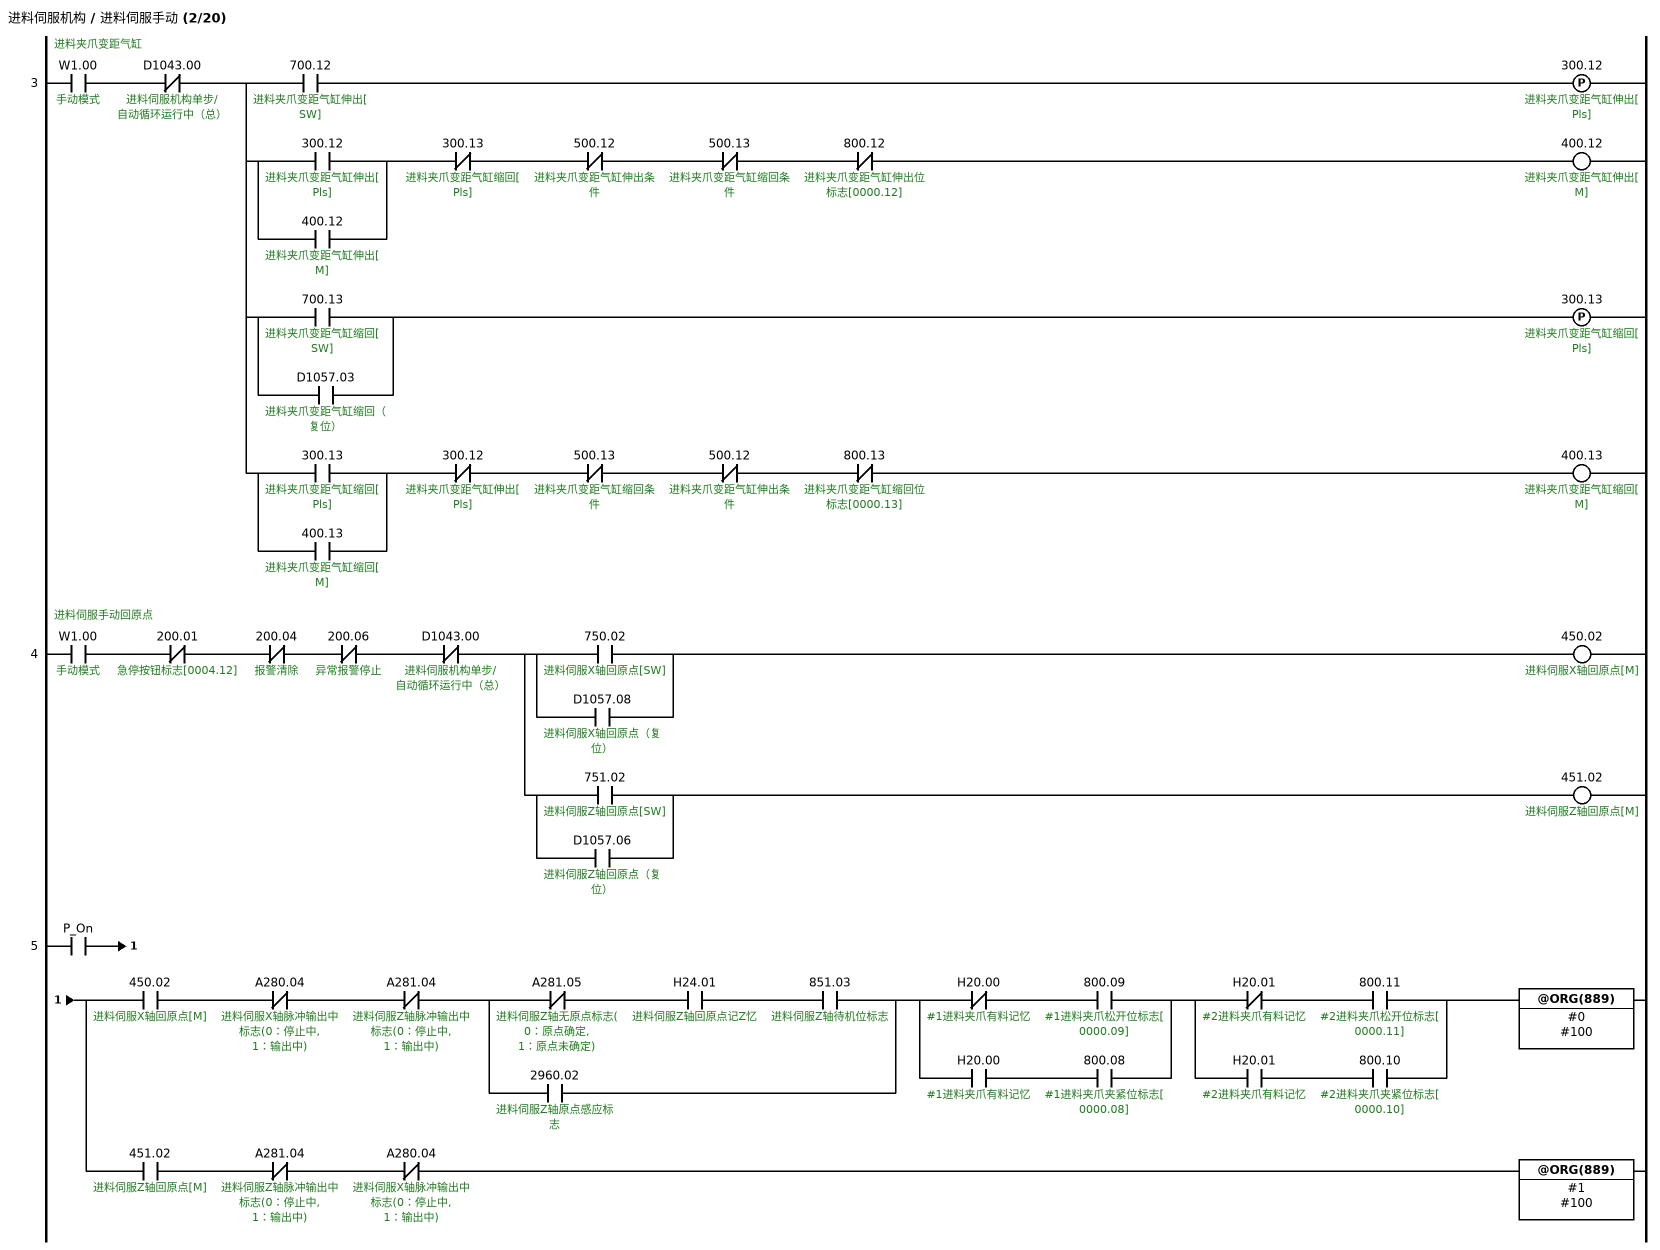
; rung 3: 进料夹爪变距气缸
LD W1.00  ; 手动模式
ANDNOT D1043.00  ; 进料伺服机构单步/自动循环运行中（总）
OUT TR0
AND 700.12  ; 进料夹爪变距气缸伸出[SW]
DIFU(013) 300.12  ; 进料夹爪变距气缸伸出[Pls]
LD TR0
LD 300.12  ; 进料夹爪变距气缸伸出[Pls]
OR 400.12  ; 进料夹爪变距气缸伸出[M]
ANDLD
ANDNOT 300.13  ; 进料夹爪变距气缸缩回[Pls]
ANDNOT 500.12  ; 进料夹爪变距气缸伸出条件
ANDNOT 500.13  ; 进料夹爪变距气缸缩回条件
ANDNOT 800.12  ; 进料夹爪变距气缸伸出位标志[0000.12]
OUT 400.12  ; 进料夹爪变距气缸伸出[M]
LD TR0
LD 700.13  ; 进料夹爪变距气缸缩回[SW]
OR D1057.03  ; 进料夹爪变距气缸缩回（复位）
ANDLD
DIFU(013) 300.13  ; 进料夹爪变距气缸缩回[Pls]
LD TR0
LD 300.13  ; 进料夹爪变距气缸缩回[Pls]
OR 400.13  ; 进料夹爪变距气缸缩回[M]
ANDLD
ANDNOT 300.12  ; 进料夹爪变距气缸伸出[Pls]
ANDNOT 500.13  ; 进料夹爪变距气缸缩回条件
ANDNOT 500.12  ; 进料夹爪变距气缸伸出条件
ANDNOT 800.13  ; 进料夹爪变距气缸缩回位标志[0000.13]
OUT 400.13  ; 进料夹爪变距气缸缩回[M]
; rung 4: 进料伺服手动回原点
LD W1.00  ; 手动模式
ANDNOT 200.01  ; 急停按钮标志[0004.12]
ANDNOT 200.04  ; 报警清除
ANDNOT 200.06  ; 异常报警停止
ANDNOT D1043.00  ; 进料伺服机构单步/自动循环运行中（总）
OUT TR0
LD 750.02  ; 进料伺服X轴回原点[SW]
OR D1057.08  ; 进料伺服X轴回原点（复位）
ANDLD
OUT 450.02  ; 进料伺服X轴回原点[M]
LD TR0
LD 751.02  ; 进料伺服Z轴回原点[SW]
OR D1057.06  ; 进料伺服Z轴回原点（复位）
ANDLD
OUT 451.02  ; 进料伺服Z轴回原点[M]
; rung 5
LD P_On
OUT TR0
AND 450.02  ; 进料伺服X轴回原点[M]
ANDNOT A280.04  ; 进料伺服X轴脉冲输出中标志(0：停止中,1：输出中)
ANDNOT A281.04  ; 进料伺服Z轴脉冲输出中标志(0：停止中,1：输出中)
LDNOT A281.05  ; 进料伺服Z轴无原点标志(0：原点确定,1：原点未确定)
AND H24.01  ; 进料伺服Z轴回原点记Z忆
AND 851.03  ; 进料伺服Z轴待机位标志
OR 2960.02  ; 进料伺服Z轴原点感应标志
ANDLD
LDNOT H20.00  ; #1进料夹爪有料记忆
AND 800.09  ; #1进料夹爪松开位标志[0000.09]
LD H20.00  ; #1进料夹爪有料记忆
AND 800.08  ; #1进料夹爪夹紧位标志[0000.08]
ORLD
ANDLD
LDNOT H20.01  ; #2进料夹爪有料记忆
AND 800.11  ; #2进料夹爪松开位标志[0000.11]
LD H20.01  ; #2进料夹爪有料记忆
AND 800.10  ; #2进料夹爪夹紧位标志[0000.10]
ORLD
ANDLD
@ORG(889) #0 #100
LD TR0
AND 451.02  ; 进料伺服Z轴回原点[M]
ANDNOT A281.04  ; 进料伺服Z轴脉冲输出中标志(0：停止中,1：输出中)
ANDNOT A280.04  ; 进料伺服X轴脉冲输出中标志(0：停止中,1：输出中)
@ORG(889) #1 #100

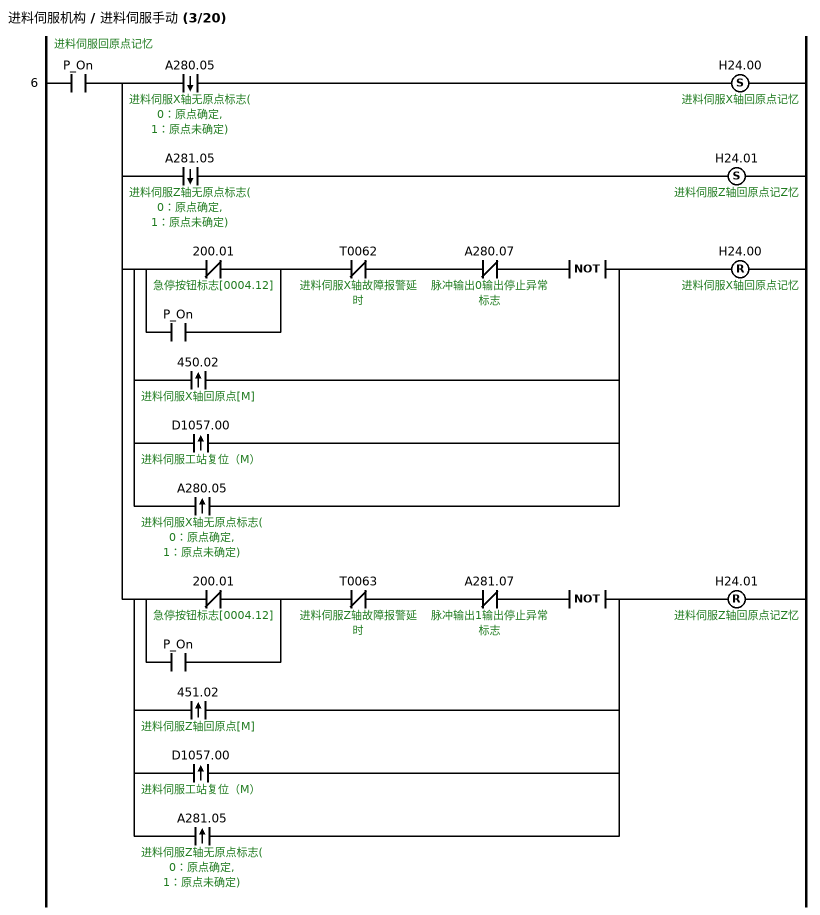
; rung 6: 进料伺服回原点记忆
LD P_On
OUT TR0
%AND A280.05  ; 进料伺服X轴无原点标志(0：原点确定,1：原点未确定)
SET H24.00  ; 进料伺服X轴回原点记忆
LD TR0
%AND A281.05  ; 进料伺服Z轴无原点标志(0：原点确定,1：原点未确定)
SET H24.01  ; 进料伺服Z轴回原点记Z忆
LD TR0
LDNOT 200.01  ; 急停按钮标志[0004.12]
OR P_On
ANDNOT T0062  ; 进料伺服X轴故障报警延时
ANDNOT A280.07  ; 脉冲输出0输出停止异常标志
NOT(520)
@OR 450.02  ; 进料伺服X轴回原点[M]
@OR D1057.00  ; 进料伺服工站复位（M）
@OR A280.05  ; 进料伺服X轴无原点标志(0：原点确定,1：原点未确定)
ANDLD
RSET H24.00  ; 进料伺服X轴回原点记忆
LD TR0
LDNOT 200.01  ; 急停按钮标志[0004.12]
OR P_On
ANDNOT T0063  ; 进料伺服Z轴故障报警延时
ANDNOT A281.07  ; 脉冲输出1输出停止异常标志
NOT(520)
@OR 451.02  ; 进料伺服Z轴回原点[M]
@OR D1057.00  ; 进料伺服工站复位（M）
@OR A281.05  ; 进料伺服Z轴无原点标志(0：原点确定,1：原点未确定)
ANDLD
RSET H24.01  ; 进料伺服Z轴回原点记Z忆

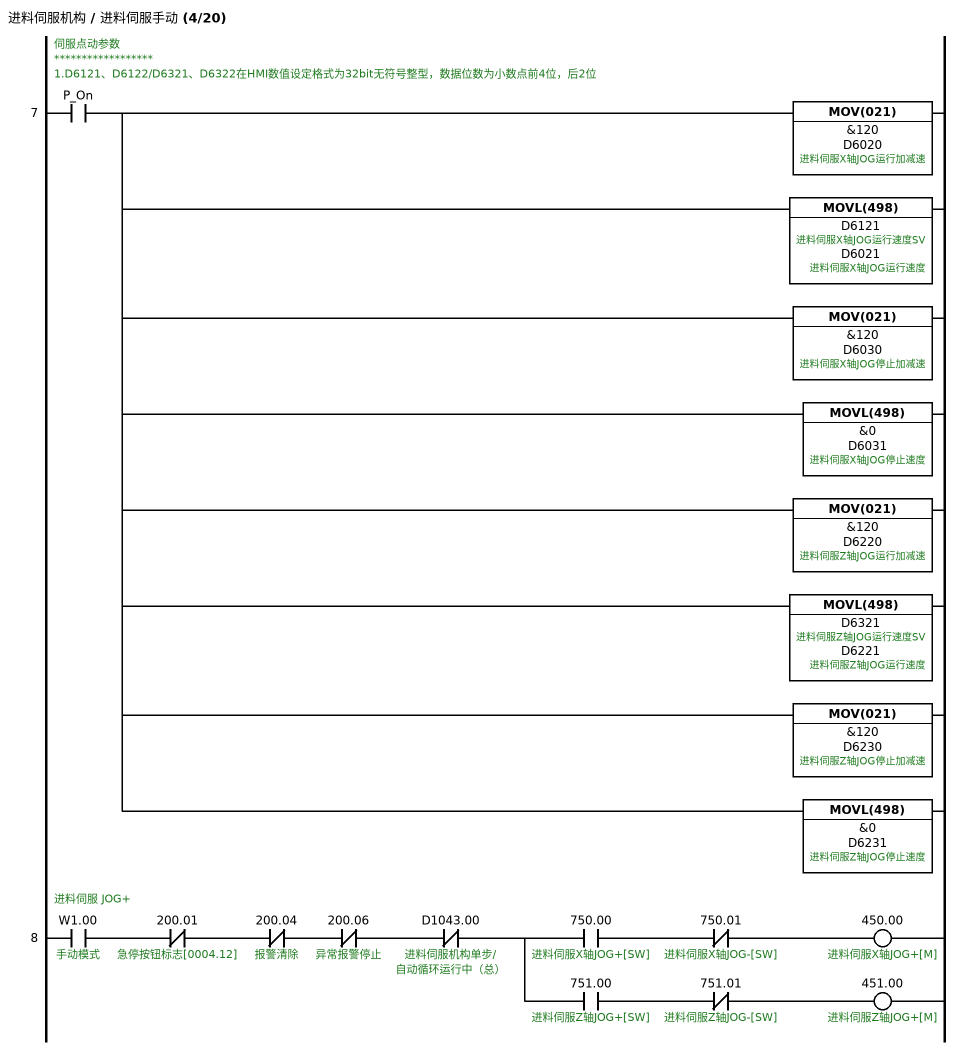
; rung 7: 伺服点动参数 / ****************** / 1.D6121、D6122/D6321、D6322在HMI数值设定格式为32bit无符号整型，数据位数为小数点前4位，后2位
LD P_On
MOV(021) &120 D6020  ; 进料伺服X轴JOG运行加减速
MOVL(498) D6121 D6021  ; 进料伺服X轴JOG运行速度SV, 进料伺服X轴JOG运行速度
MOV(021) &120 D6030  ; 进料伺服X轴JOG停止加减速
MOVL(498) &0 D6031  ; 进料伺服X轴JOG停止速度
MOV(021) &120 D6220  ; 进料伺服Z轴JOG运行加减速
MOVL(498) D6321 D6221  ; 进料伺服Z轴JOG运行速度SV, 进料伺服Z轴JOG运行速度
MOV(021) &120 D6230  ; 进料伺服Z轴JOG停止加减速
MOVL(498) &0 D6231  ; 进料伺服Z轴JOG停止速度
; rung 8: 进料伺服 JOG+
LD W1.00  ; 手动模式
ANDNOT 200.01  ; 急停按钮标志[0004.12]
ANDNOT 200.04  ; 报警清除
ANDNOT 200.06  ; 异常报警停止
ANDNOT D1043.00  ; 进料伺服机构单步/自动循环运行中（总）
OUT TR0
AND 750.00  ; 进料伺服X轴JOG+[SW]
ANDNOT 750.01  ; 进料伺服X轴JOG-[SW]
OUT 450.00  ; 进料伺服X轴JOG+[M]
LD TR0
AND 751.00  ; 进料伺服Z轴JOG+[SW]
ANDNOT 751.01  ; 进料伺服Z轴JOG-[SW]
OUT 451.00  ; 进料伺服Z轴JOG+[M]

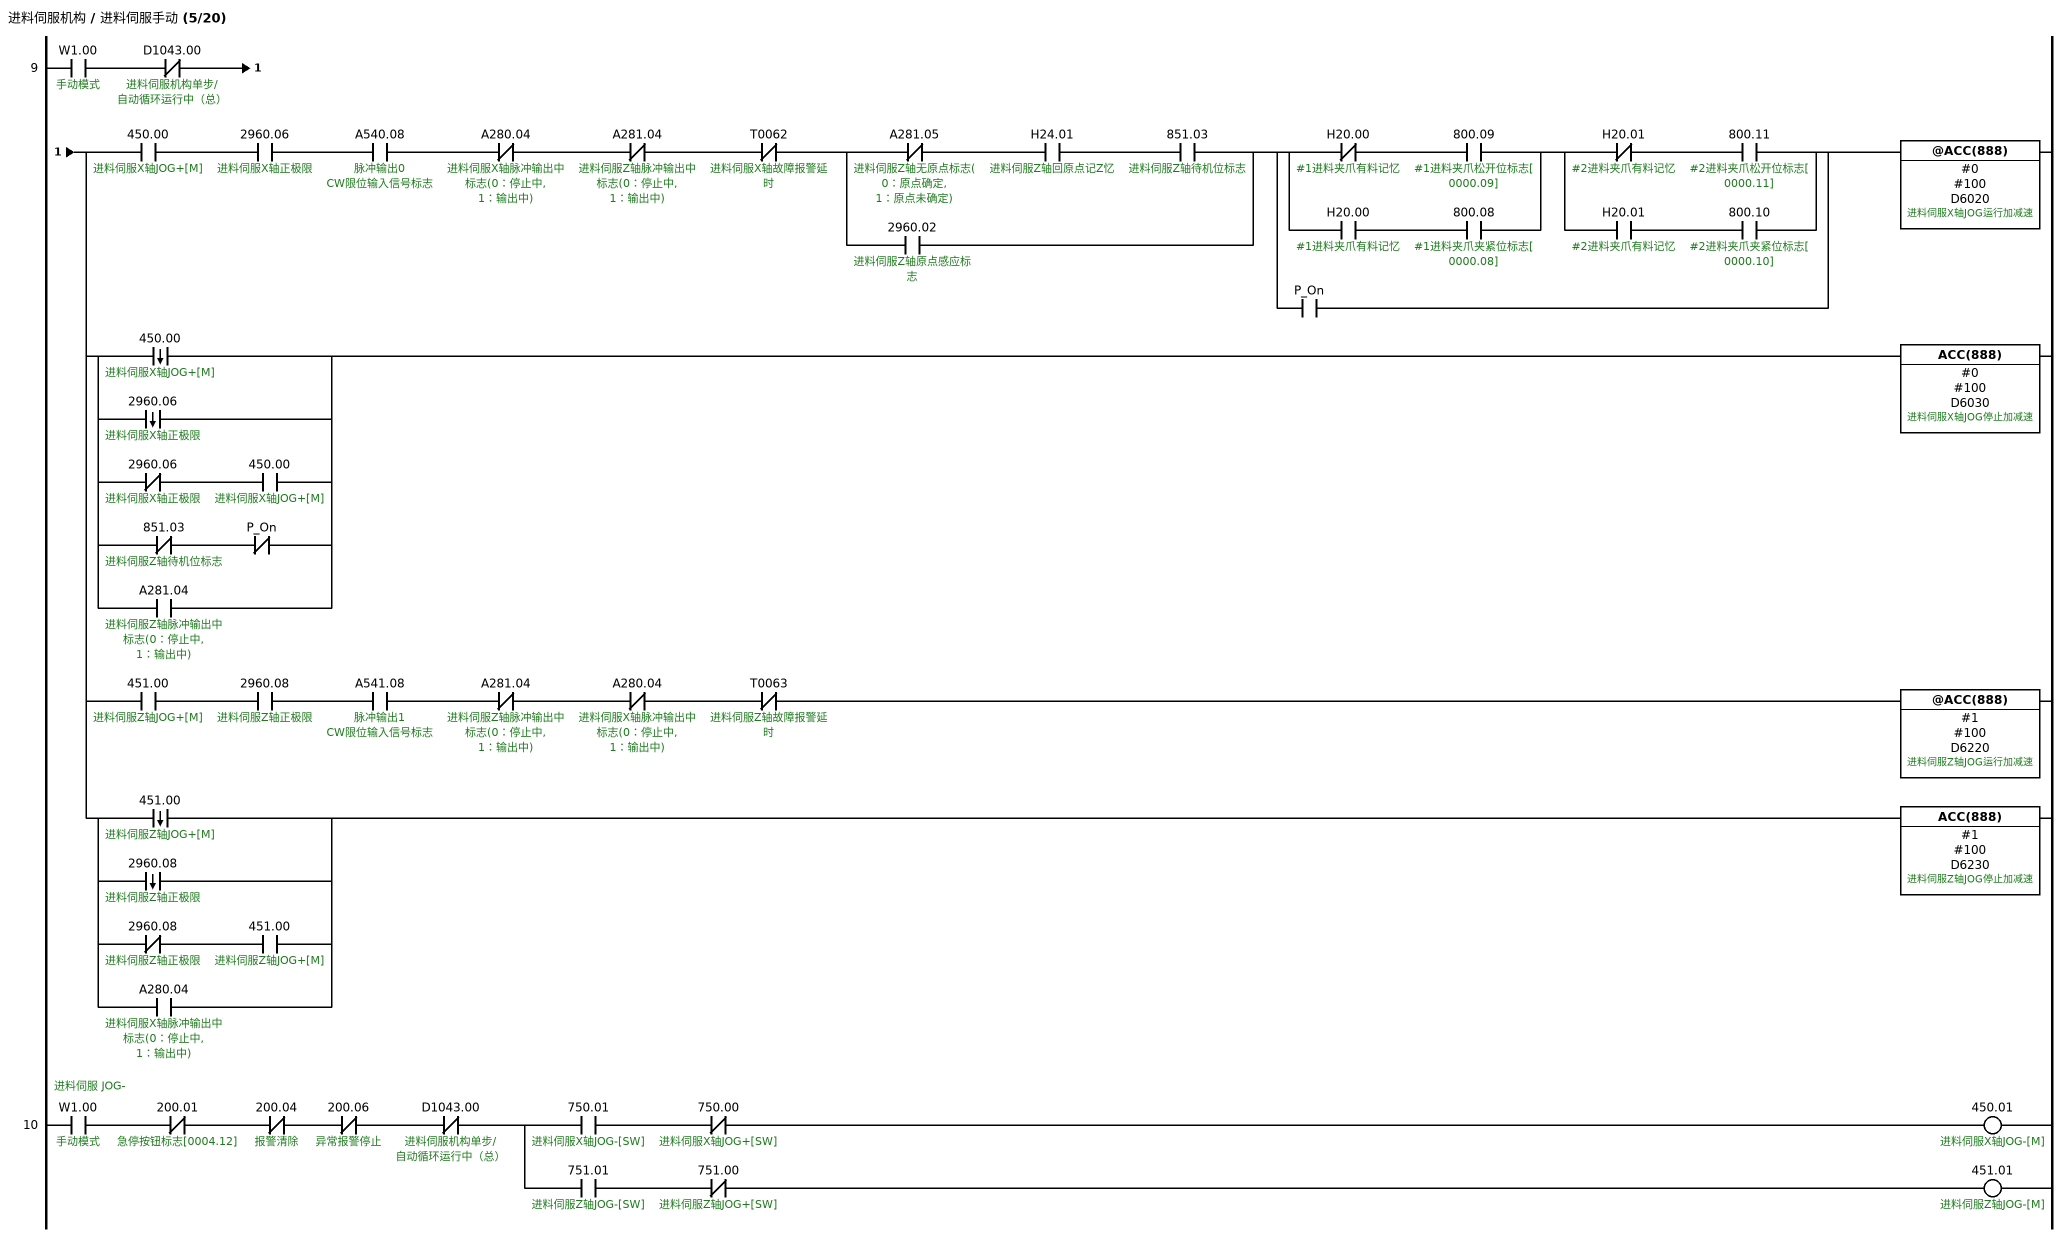
; rung 9
LD W1.00  ; 手动模式
ANDNOT D1043.00  ; 进料伺服机构单步/自动循环运行中（总）
OUT TR0
AND 450.00  ; 进料伺服X轴JOG+[M]
AND 2960.06  ; 进料伺服X轴正极限
AND A540.08  ; 脉冲输出0 CW限位输入信号标志
ANDNOT A280.04  ; 进料伺服X轴脉冲输出中标志(0：停止中,1：输出中)
ANDNOT A281.04  ; 进料伺服Z轴脉冲输出中标志(0：停止中,1：输出中)
ANDNOT T0062  ; 进料伺服X轴故障报警延时
LDNOT A281.05  ; 进料伺服Z轴无原点标志(0：原点确定,1：原点未确定)
AND H24.01  ; 进料伺服Z轴回原点记Z忆
AND 851.03  ; 进料伺服Z轴待机位标志
OR 2960.02  ; 进料伺服Z轴原点感应标志
ANDLD
LDNOT H20.00  ; #1进料夹爪有料记忆
AND 800.09  ; #1进料夹爪松开位标志[0000.09]
LD H20.00  ; #1进料夹爪有料记忆
AND 800.08  ; #1进料夹爪夹紧位标志[0000.08]
ORLD
LDNOT H20.01  ; #2进料夹爪有料记忆
AND 800.11  ; #2进料夹爪松开位标志[0000.11]
LD H20.01  ; #2进料夹爪有料记忆
AND 800.10  ; #2进料夹爪夹紧位标志[0000.10]
ORLD
ANDLD
OR P_On
ANDLD
@ACC(888) #0 #100 D6020  ; 进料伺服X轴JOG运行加减速
LD TR0
%LD 450.00  ; 进料伺服X轴JOG+[M]
%OR 2960.06  ; 进料伺服X轴正极限
LDNOT 2960.06  ; 进料伺服X轴正极限
AND 450.00  ; 进料伺服X轴JOG+[M]
ORLD
LDNOT 851.03  ; 进料伺服Z轴待机位标志
ANDNOT P_On
ORLD
OR A281.04  ; 进料伺服Z轴脉冲输出中标志(0：停止中,1：输出中)
ANDLD
ACC(888) #0 #100 D6030  ; 进料伺服X轴JOG停止加减速
LD TR0
AND 451.00  ; 进料伺服Z轴JOG+[M]
AND 2960.08  ; 进料伺服Z轴正极限
AND A541.08  ; 脉冲输出1 CW限位输入信号标志
ANDNOT A281.04  ; 进料伺服Z轴脉冲输出中标志(0：停止中,1：输出中)
ANDNOT A280.04  ; 进料伺服X轴脉冲输出中标志(0：停止中,1：输出中)
ANDNOT T0063  ; 进料伺服Z轴故障报警延时
@ACC(888) #1 #100 D6220  ; 进料伺服Z轴JOG运行加减速
LD TR0
%LD 451.00  ; 进料伺服Z轴JOG+[M]
%OR 2960.08  ; 进料伺服Z轴正极限
LDNOT 2960.08  ; 进料伺服Z轴正极限
AND 451.00  ; 进料伺服Z轴JOG+[M]
ORLD
OR A280.04  ; 进料伺服X轴脉冲输出中标志(0：停止中,1：输出中)
ANDLD
ACC(888) #1 #100 D6230  ; 进料伺服Z轴JOG停止加减速
; rung 10: 进料伺服 JOG-
LD W1.00  ; 手动模式
ANDNOT 200.01  ; 急停按钮标志[0004.12]
ANDNOT 200.04  ; 报警清除
ANDNOT 200.06  ; 异常报警停止
ANDNOT D1043.00  ; 进料伺服机构单步/自动循环运行中（总）
OUT TR0
AND 750.01  ; 进料伺服X轴JOG-[SW]
ANDNOT 750.00  ; 进料伺服X轴JOG+[SW]
OUT 450.01  ; 进料伺服X轴JOG-[M]
LD TR0
AND 751.01  ; 进料伺服Z轴JOG-[SW]
ANDNOT 751.00  ; 进料伺服Z轴JOG+[SW]
OUT 451.01  ; 进料伺服Z轴JOG-[M]

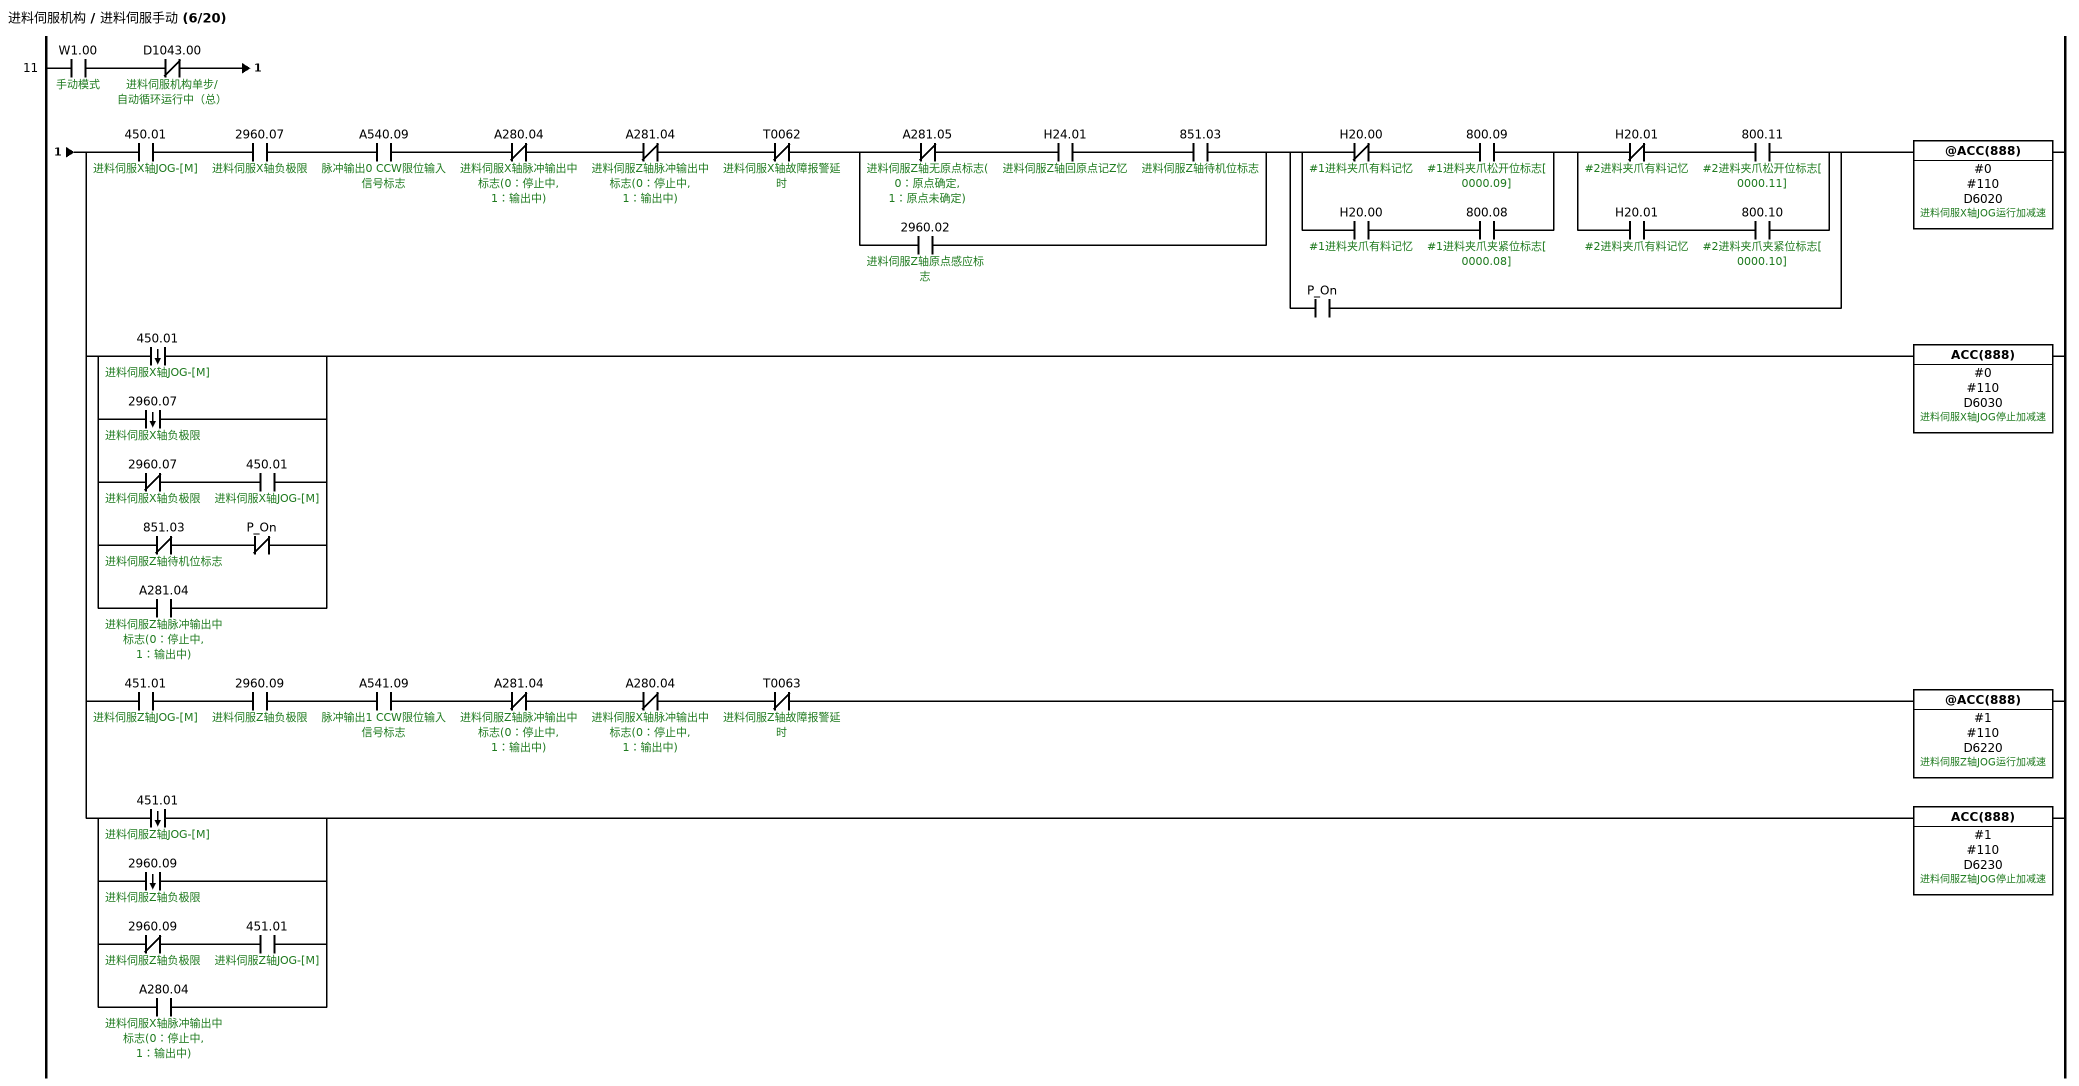
; rung 11
LD W1.00  ; 手动模式
ANDNOT D1043.00  ; 进料伺服机构单步/自动循环运行中（总）
OUT TR0
AND 450.01  ; 进料伺服X轴JOG-[M]
AND 2960.07  ; 进料伺服X轴负极限
AND A540.09  ; 脉冲输出0 CCW限位输入信号标志
ANDNOT A280.04  ; 进料伺服X轴脉冲输出中标志(0：停止中,1：输出中)
ANDNOT A281.04  ; 进料伺服Z轴脉冲输出中标志(0：停止中,1：输出中)
ANDNOT T0062  ; 进料伺服X轴故障报警延时
LDNOT A281.05  ; 进料伺服Z轴无原点标志(0：原点确定,1：原点未确定)
AND H24.01  ; 进料伺服Z轴回原点记Z忆
AND 851.03  ; 进料伺服Z轴待机位标志
OR 2960.02  ; 进料伺服Z轴原点感应标志
ANDLD
LDNOT H20.00  ; #1进料夹爪有料记忆
AND 800.09  ; #1进料夹爪松开位标志[0000.09]
LD H20.00  ; #1进料夹爪有料记忆
AND 800.08  ; #1进料夹爪夹紧位标志[0000.08]
ORLD
LDNOT H20.01  ; #2进料夹爪有料记忆
AND 800.11  ; #2进料夹爪松开位标志[0000.11]
LD H20.01  ; #2进料夹爪有料记忆
AND 800.10  ; #2进料夹爪夹紧位标志[0000.10]
ORLD
ANDLD
OR P_On
ANDLD
@ACC(888) #0 #110 D6020  ; 进料伺服X轴JOG运行加减速
LD TR0
%LD 450.01  ; 进料伺服X轴JOG-[M]
%OR 2960.07  ; 进料伺服X轴负极限
LDNOT 2960.07  ; 进料伺服X轴负极限
AND 450.01  ; 进料伺服X轴JOG-[M]
ORLD
LDNOT 851.03  ; 进料伺服Z轴待机位标志
ANDNOT P_On
ORLD
OR A281.04  ; 进料伺服Z轴脉冲输出中标志(0：停止中,1：输出中)
ANDLD
ACC(888) #0 #110 D6030  ; 进料伺服X轴JOG停止加减速
LD TR0
AND 451.01  ; 进料伺服Z轴JOG-[M]
AND 2960.09  ; 进料伺服Z轴负极限
AND A541.09  ; 脉冲输出1 CCW限位输入信号标志
ANDNOT A281.04  ; 进料伺服Z轴脉冲输出中标志(0：停止中,1：输出中)
ANDNOT A280.04  ; 进料伺服X轴脉冲输出中标志(0：停止中,1：输出中)
ANDNOT T0063  ; 进料伺服Z轴故障报警延时
@ACC(888) #1 #110 D6220  ; 进料伺服Z轴JOG运行加减速
LD TR0
%LD 451.01  ; 进料伺服Z轴JOG-[M]
%OR 2960.09  ; 进料伺服Z轴负极限
LDNOT 2960.09  ; 进料伺服Z轴负极限
AND 451.01  ; 进料伺服Z轴JOG-[M]
ORLD
OR A280.04  ; 进料伺服X轴脉冲输出中标志(0：停止中,1：输出中)
ANDLD
ACC(888) #1 #110 D6230  ; 进料伺服Z轴JOG停止加减速

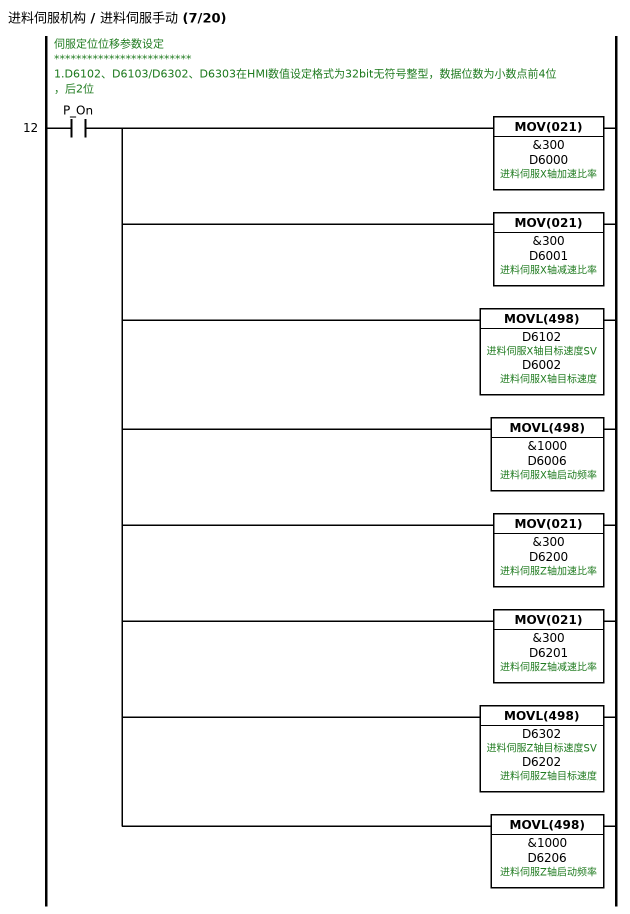
; rung 12: 伺服定位位移参数设定 / ************************* / 1.D6102、D6103/D6302、D6303在HMI数值设定格式为32bit无符号整型，数据位数为小数点前4位，后2位
LD P_On
MOV(021) &300 D6000  ; 进料伺服X轴加速比率
MOV(021) &300 D6001  ; 进料伺服X轴减速比率
MOVL(498) D6102 D6002  ; 进料伺服X轴目标速度SV, 进料伺服X轴目标速度
MOVL(498) &1000 D6006  ; 进料伺服X轴启动频率
MOV(021) &300 D6200  ; 进料伺服Z轴加速比率
MOV(021) &300 D6201  ; 进料伺服Z轴减速比率
MOVL(498) D6302 D6202  ; 进料伺服Z轴目标速度SV, 进料伺服Z轴目标速度
MOVL(498) &1000 D6206  ; 进料伺服Z轴启动频率

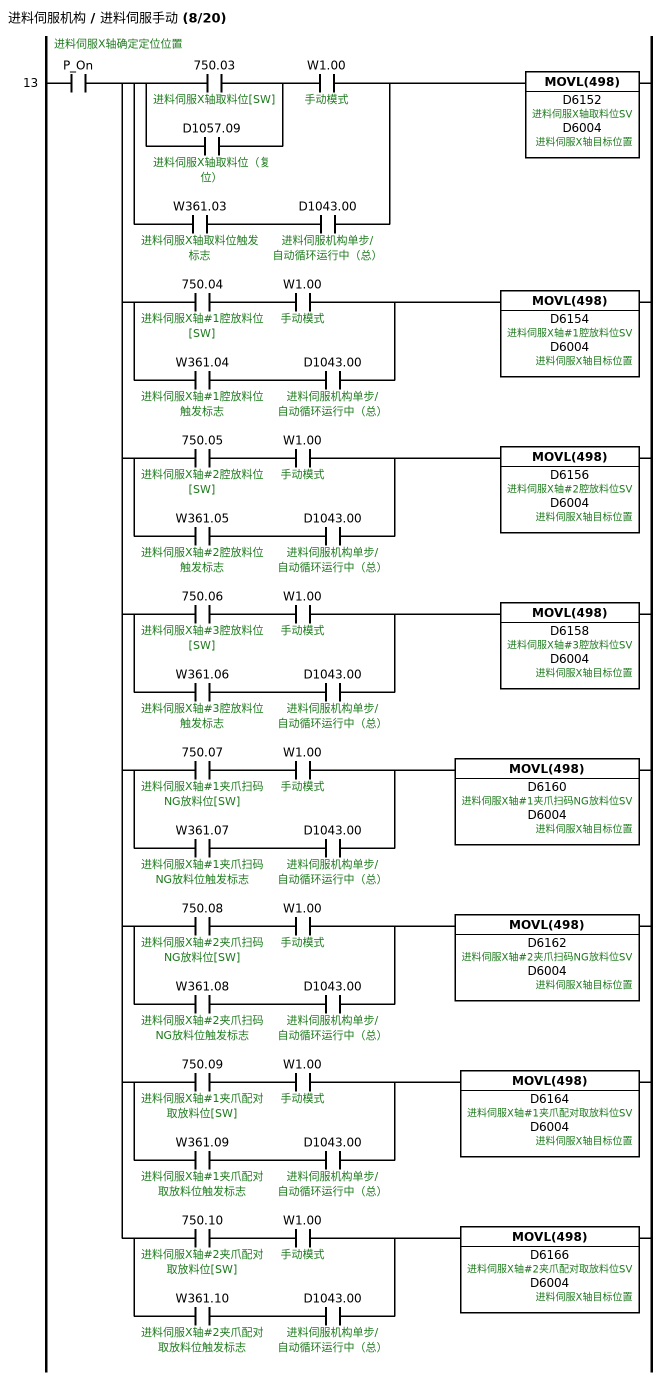
; rung 13: 进料伺服X轴确定定位位置
LD P_On
OUT TR0
LD 750.03  ; 进料伺服X轴取料位[SW]
OR D1057.09  ; 进料伺服X轴取料位（复位）
AND W1.00  ; 手动模式
LD W361.03  ; 进料伺服X轴取料位触发标志
AND D1043.00  ; 进料伺服机构单步/自动循环运行中（总）
ORLD
ANDLD
MOVL(498) D6152 D6004  ; 进料伺服X轴取料位SV, 进料伺服X轴目标位置
LD TR0
LD 750.04  ; 进料伺服X轴#1腔放料位[SW]
AND W1.00  ; 手动模式
LD W361.04  ; 进料伺服X轴#1腔放料位触发标志
AND D1043.00  ; 进料伺服机构单步/自动循环运行中（总）
ORLD
ANDLD
MOVL(498) D6154 D6004  ; 进料伺服X轴#1腔放料位SV, 进料伺服X轴目标位置
LD TR0
LD 750.05  ; 进料伺服X轴#2腔放料位[SW]
AND W1.00  ; 手动模式
LD W361.05  ; 进料伺服X轴#2腔放料位触发标志
AND D1043.00  ; 进料伺服机构单步/自动循环运行中（总）
ORLD
ANDLD
MOVL(498) D6156 D6004  ; 进料伺服X轴#2腔放料位SV, 进料伺服X轴目标位置
LD TR0
LD 750.06  ; 进料伺服X轴#3腔放料位[SW]
AND W1.00  ; 手动模式
LD W361.06  ; 进料伺服X轴#3腔放料位触发标志
AND D1043.00  ; 进料伺服机构单步/自动循环运行中（总）
ORLD
ANDLD
MOVL(498) D6158 D6004  ; 进料伺服X轴#3腔放料位SV, 进料伺服X轴目标位置
LD TR0
LD 750.07  ; 进料伺服X轴#1夹爪扫码NG放料位[SW]
AND W1.00  ; 手动模式
LD W361.07  ; 进料伺服X轴#1夹爪扫码NG放料位触发标志
AND D1043.00  ; 进料伺服机构单步/自动循环运行中（总）
ORLD
ANDLD
MOVL(498) D6160 D6004  ; 进料伺服X轴#1夹爪扫码NG放料位SV, 进料伺服X轴目标位置
LD TR0
LD 750.08  ; 进料伺服X轴#2夹爪扫码NG放料位[SW]
AND W1.00  ; 手动模式
LD W361.08  ; 进料伺服X轴#2夹爪扫码NG放料位触发标志
AND D1043.00  ; 进料伺服机构单步/自动循环运行中（总）
ORLD
ANDLD
MOVL(498) D6162 D6004  ; 进料伺服X轴#2夹爪扫码NG放料位SV, 进料伺服X轴目标位置
LD TR0
LD 750.09  ; 进料伺服X轴#1夹爪配对取放料位[SW]
AND W1.00  ; 手动模式
LD W361.09  ; 进料伺服X轴#1夹爪配对取放料位触发标志
AND D1043.00  ; 进料伺服机构单步/自动循环运行中（总）
ORLD
ANDLD
MOVL(498) D6164 D6004  ; 进料伺服X轴#1夹爪配对取放料位SV, 进料伺服X轴目标位置
LD TR0
LD 750.10  ; 进料伺服X轴#2夹爪配对取放料位[SW]
AND W1.00  ; 手动模式
LD W361.10  ; 进料伺服X轴#2夹爪配对取放料位触发标志
AND D1043.00  ; 进料伺服机构单步/自动循环运行中（总）
ORLD
ANDLD
MOVL(498) D6166 D6004  ; 进料伺服X轴#2夹爪配对取放料位SV, 进料伺服X轴目标位置

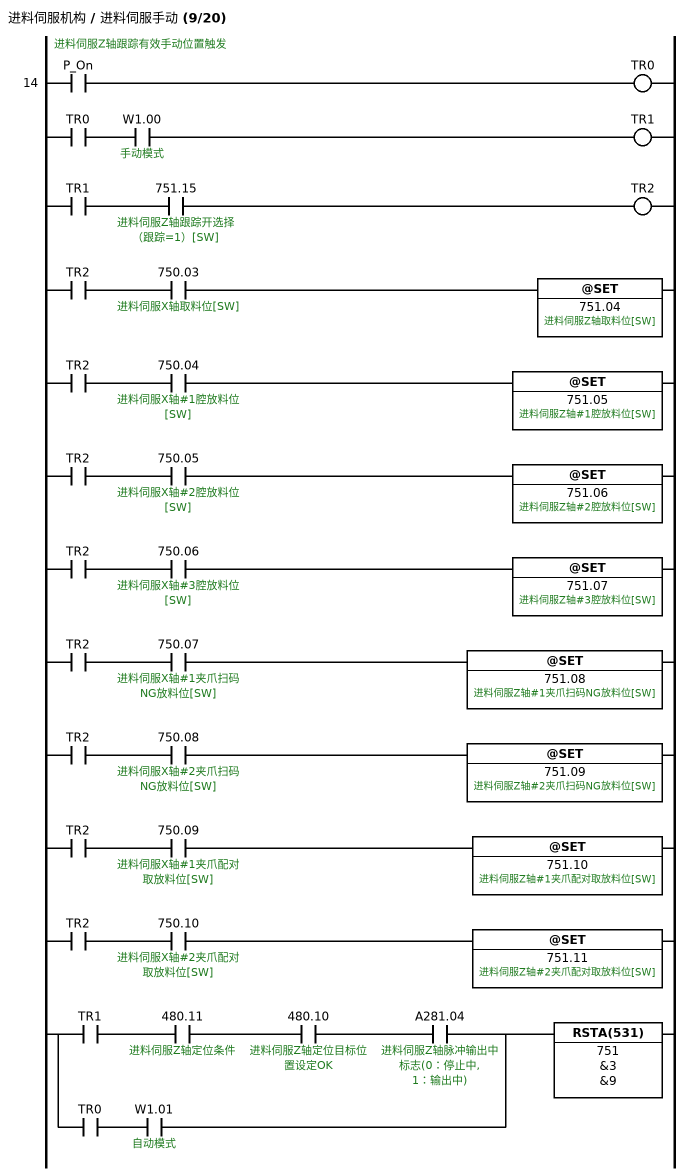
; rung 14: 进料伺服Z轴跟踪有效手动位置触发
LD P_On
OUT TR0
AND W1.00  ; 手动模式
OUT TR1
AND 751.15  ; 进料伺服Z轴跟踪开选择（跟踪=1）[SW]
OUT TR2
AND 750.03  ; 进料伺服X轴取料位[SW]
@SET 751.04  ; 进料伺服Z轴取料位[SW]
LD TR2
AND 750.04  ; 进料伺服X轴#1腔放料位[SW]
@SET 751.05  ; 进料伺服Z轴#1腔放料位[SW]
LD TR2
AND 750.05  ; 进料伺服X轴#2腔放料位[SW]
@SET 751.06  ; 进料伺服Z轴#2腔放料位[SW]
LD TR2
AND 750.06  ; 进料伺服X轴#3腔放料位[SW]
@SET 751.07  ; 进料伺服Z轴#3腔放料位[SW]
LD TR2
AND 750.07  ; 进料伺服X轴#1夹爪扫码NG放料位[SW]
@SET 751.08  ; 进料伺服Z轴#1夹爪扫码NG放料位[SW]
LD TR2
AND 750.08  ; 进料伺服X轴#2夹爪扫码NG放料位[SW]
@SET 751.09  ; 进料伺服Z轴#2夹爪扫码NG放料位[SW]
LD TR2
AND 750.09  ; 进料伺服X轴#1夹爪配对取放料位[SW]
@SET 751.10  ; 进料伺服Z轴#1夹爪配对取放料位[SW]
LD TR2
AND 750.10  ; 进料伺服X轴#2夹爪配对取放料位[SW]
@SET 751.11  ; 进料伺服Z轴#2夹爪配对取放料位[SW]
LD TR1
AND 480.11  ; 进料伺服Z轴定位条件
AND 480.10  ; 进料伺服Z轴定位目标位置设定OK
AND A281.04  ; 进料伺服Z轴脉冲输出中标志(0：停止中,1：输出中)
LD TR0
AND W1.01  ; 自动模式
ORLD
RSTA(531) 751 &3 &9

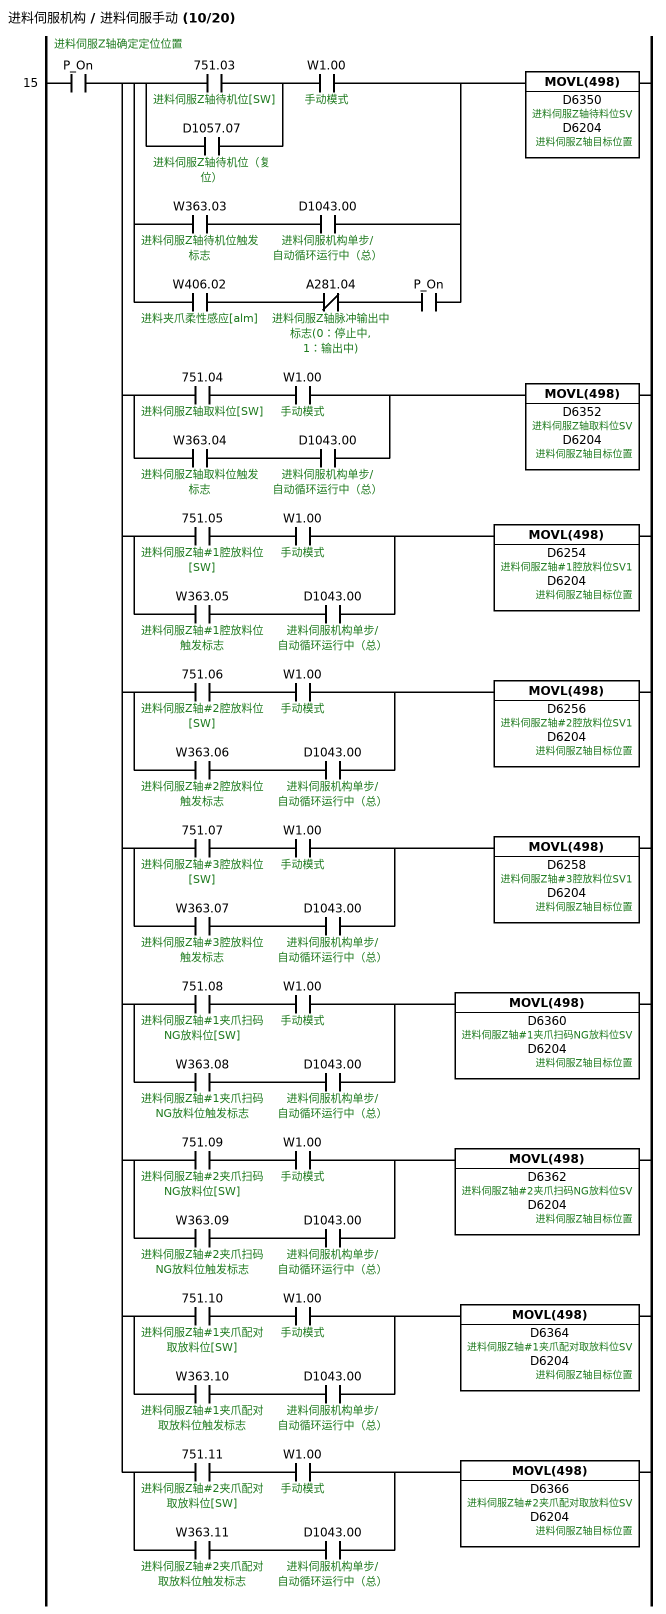
; rung 15: 进料伺服Z轴确定定位位置
LD P_On
OUT TR0
LD 751.03  ; 进料伺服Z轴待机位[SW]
OR D1057.07  ; 进料伺服Z轴待机位（复位）
AND W1.00  ; 手动模式
LD W363.03  ; 进料伺服Z轴待机位触发标志
AND D1043.00  ; 进料伺服机构单步/自动循环运行中（总）
ORLD
LD W406.02  ; 进料夹爪柔性感应[alm]
ANDNOT A281.04  ; 进料伺服Z轴脉冲输出中标志(0：停止中,1：输出中)
AND P_On
ORLD
ANDLD
MOVL(498) D6350 D6204  ; 进料伺服Z轴待料位SV, 进料伺服Z轴目标位置
LD TR0
LD 751.04  ; 进料伺服Z轴取料位[SW]
AND W1.00  ; 手动模式
LD W363.04  ; 进料伺服Z轴取料位触发标志
AND D1043.00  ; 进料伺服机构单步/自动循环运行中（总）
ORLD
ANDLD
MOVL(498) D6352 D6204  ; 进料伺服Z轴取料位SV, 进料伺服Z轴目标位置
LD TR0
LD 751.05  ; 进料伺服Z轴#1腔放料位[SW]
AND W1.00  ; 手动模式
LD W363.05  ; 进料伺服Z轴#1腔放料位触发标志
AND D1043.00  ; 进料伺服机构单步/自动循环运行中（总）
ORLD
ANDLD
MOVL(498) D6254 D6204  ; 进料伺服Z轴#1腔放料位SV1, 进料伺服Z轴目标位置
LD TR0
LD 751.06  ; 进料伺服Z轴#2腔放料位[SW]
AND W1.00  ; 手动模式
LD W363.06  ; 进料伺服Z轴#2腔放料位触发标志
AND D1043.00  ; 进料伺服机构单步/自动循环运行中（总）
ORLD
ANDLD
MOVL(498) D6256 D6204  ; 进料伺服Z轴#2腔放料位SV1, 进料伺服Z轴目标位置
LD TR0
LD 751.07  ; 进料伺服Z轴#3腔放料位[SW]
AND W1.00  ; 手动模式
LD W363.07  ; 进料伺服Z轴#3腔放料位触发标志
AND D1043.00  ; 进料伺服机构单步/自动循环运行中（总）
ORLD
ANDLD
MOVL(498) D6258 D6204  ; 进料伺服Z轴#3腔放料位SV1, 进料伺服Z轴目标位置
LD TR0
LD 751.08  ; 进料伺服Z轴#1夹爪扫码NG放料位[SW]
AND W1.00  ; 手动模式
LD W363.08  ; 进料伺服Z轴#1夹爪扫码NG放料位触发标志
AND D1043.00  ; 进料伺服机构单步/自动循环运行中（总）
ORLD
ANDLD
MOVL(498) D6360 D6204  ; 进料伺服Z轴#1夹爪扫码NG放料位SV, 进料伺服Z轴目标位置
LD TR0
LD 751.09  ; 进料伺服Z轴#2夹爪扫码NG放料位[SW]
AND W1.00  ; 手动模式
LD W363.09  ; 进料伺服Z轴#2夹爪扫码NG放料位触发标志
AND D1043.00  ; 进料伺服机构单步/自动循环运行中（总）
ORLD
ANDLD
MOVL(498) D6362 D6204  ; 进料伺服Z轴#2夹爪扫码NG放料位SV, 进料伺服Z轴目标位置
LD TR0
LD 751.10  ; 进料伺服Z轴#1夹爪配对取放料位[SW]
AND W1.00  ; 手动模式
LD W363.10  ; 进料伺服Z轴#1夹爪配对取放料位触发标志
AND D1043.00  ; 进料伺服机构单步/自动循环运行中（总）
ORLD
ANDLD
MOVL(498) D6364 D6204  ; 进料伺服Z轴#1夹爪配对取放料位SV, 进料伺服Z轴目标位置
LD TR0
LD 751.11  ; 进料伺服Z轴#2夹爪配对取放料位[SW]
AND W1.00  ; 手动模式
LD W363.11  ; 进料伺服Z轴#2夹爪配对取放料位触发标志
AND D1043.00  ; 进料伺服机构单步/自动循环运行中（总）
ORLD
ANDLD
MOVL(498) D6366 D6204  ; 进料伺服Z轴#2夹爪配对取放料位SV, 进料伺服Z轴目标位置

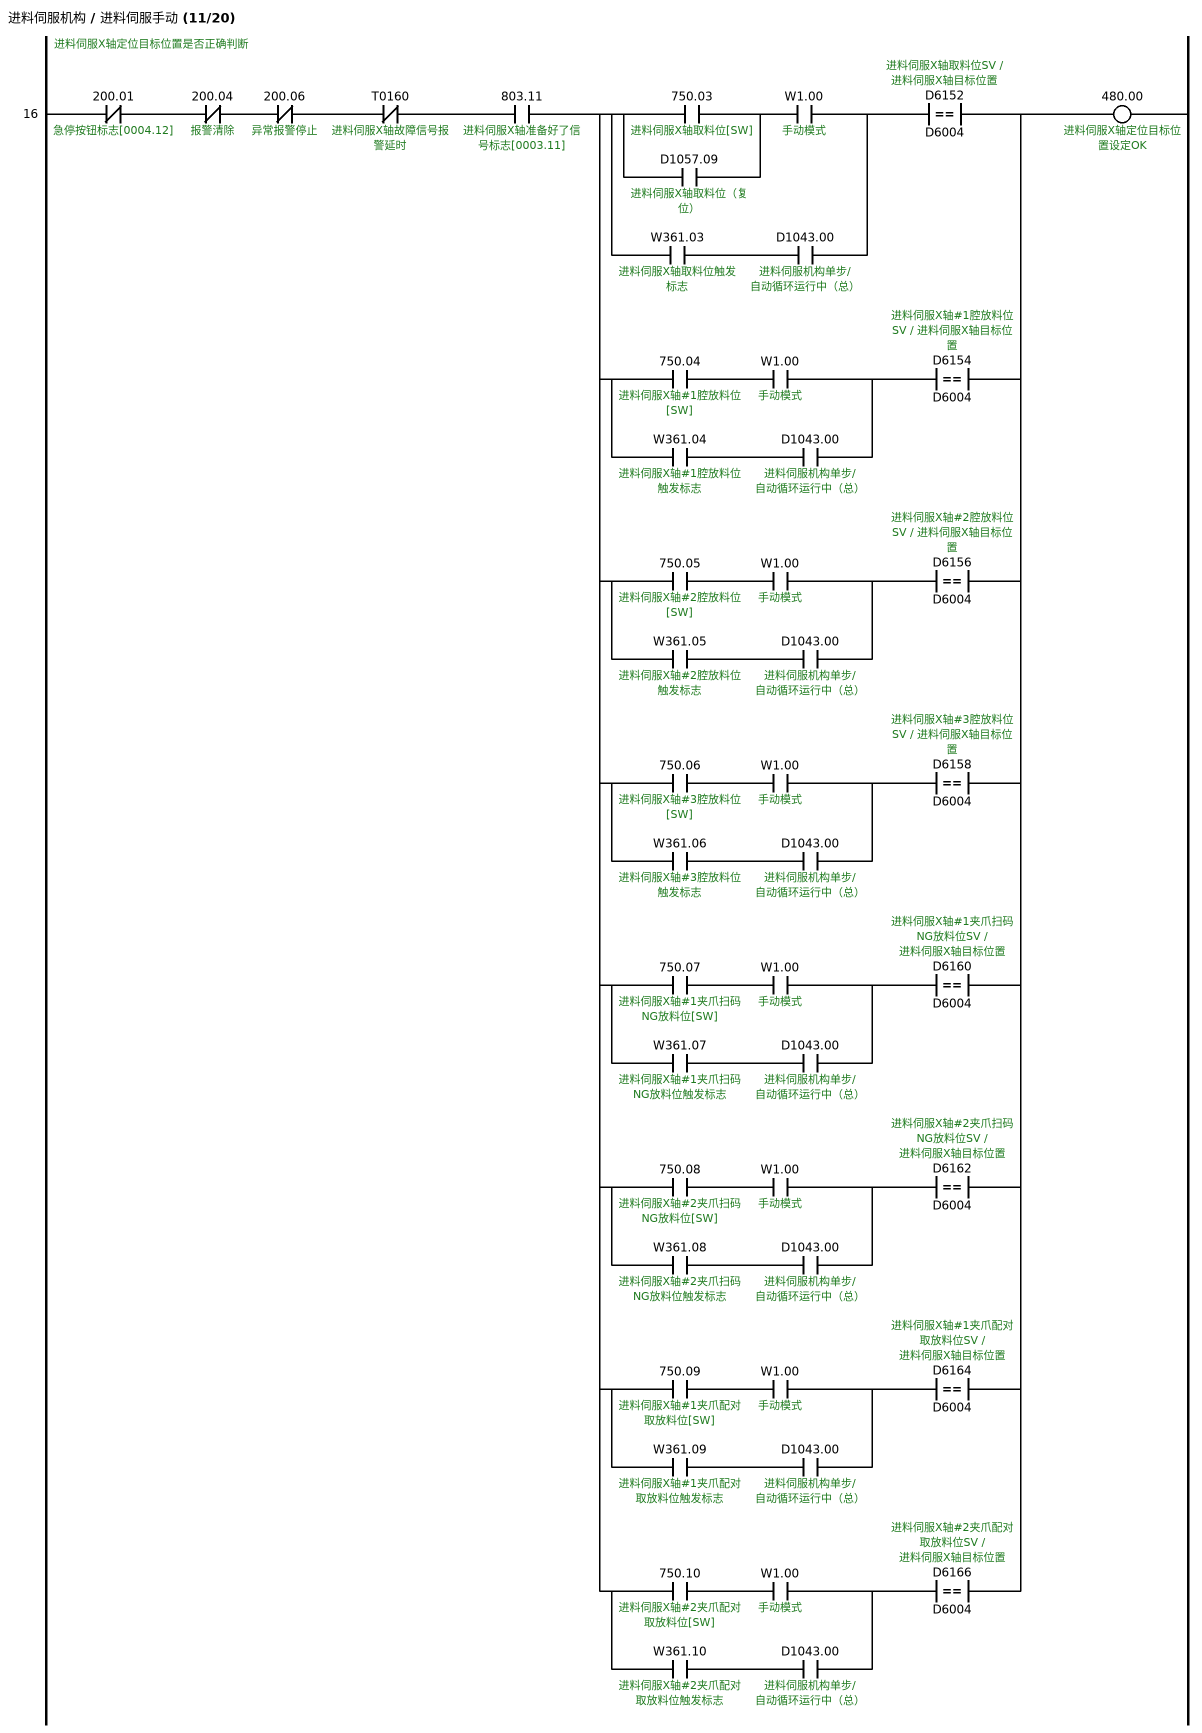
; rung 16: 进料伺服X轴定位目标位置是否正确判断
LDNOT 200.01  ; 急停按钮标志[0004.12]
ANDNOT 200.04  ; 报警清除
ANDNOT 200.06  ; 异常报警停止
ANDNOT T0160  ; 进料伺服X轴故障信号报警延时
AND 803.11  ; 进料伺服X轴准备好了信号标志[0003.11]
LD 750.03  ; 进料伺服X轴取料位[SW]
OR D1057.09  ; 进料伺服X轴取料位（复位）
AND W1.00  ; 手动模式
LD W361.03  ; 进料伺服X轴取料位触发标志
AND D1043.00  ; 进料伺服机构单步/自动循环运行中（总）
ORLD
AND=SL(303) D6152 D6004  ; 进料伺服X轴取料位SV, 进料伺服X轴目标位置
LD 750.04  ; 进料伺服X轴#1腔放料位[SW]
AND W1.00  ; 手动模式
LD W361.04  ; 进料伺服X轴#1腔放料位触发标志
AND D1043.00  ; 进料伺服机构单步/自动循环运行中（总）
ORLD
AND=SL(303) D6154 D6004  ; 进料伺服X轴#1腔放料位SV, 进料伺服X轴目标位置
ORLD
LD 750.05  ; 进料伺服X轴#2腔放料位[SW]
AND W1.00  ; 手动模式
LD W361.05  ; 进料伺服X轴#2腔放料位触发标志
AND D1043.00  ; 进料伺服机构单步/自动循环运行中（总）
ORLD
AND=SL(303) D6156 D6004  ; 进料伺服X轴#2腔放料位SV, 进料伺服X轴目标位置
ORLD
LD 750.06  ; 进料伺服X轴#3腔放料位[SW]
AND W1.00  ; 手动模式
LD W361.06  ; 进料伺服X轴#3腔放料位触发标志
AND D1043.00  ; 进料伺服机构单步/自动循环运行中（总）
ORLD
AND=SL(303) D6158 D6004  ; 进料伺服X轴#3腔放料位SV, 进料伺服X轴目标位置
ORLD
LD 750.07  ; 进料伺服X轴#1夹爪扫码NG放料位[SW]
AND W1.00  ; 手动模式
LD W361.07  ; 进料伺服X轴#1夹爪扫码NG放料位触发标志
AND D1043.00  ; 进料伺服机构单步/自动循环运行中（总）
ORLD
AND=SL(303) D6160 D6004  ; 进料伺服X轴#1夹爪扫码NG放料位SV, 进料伺服X轴目标位置
ORLD
LD 750.08  ; 进料伺服X轴#2夹爪扫码NG放料位[SW]
AND W1.00  ; 手动模式
LD W361.08  ; 进料伺服X轴#2夹爪扫码NG放料位触发标志
AND D1043.00  ; 进料伺服机构单步/自动循环运行中（总）
ORLD
AND=SL(303) D6162 D6004  ; 进料伺服X轴#2夹爪扫码NG放料位SV, 进料伺服X轴目标位置
ORLD
LD 750.09  ; 进料伺服X轴#1夹爪配对取放料位[SW]
AND W1.00  ; 手动模式
LD W361.09  ; 进料伺服X轴#1夹爪配对取放料位触发标志
AND D1043.00  ; 进料伺服机构单步/自动循环运行中（总）
ORLD
AND=SL(303) D6164 D6004  ; 进料伺服X轴#1夹爪配对取放料位SV, 进料伺服X轴目标位置
ORLD
LD 750.10  ; 进料伺服X轴#2夹爪配对取放料位[SW]
AND W1.00  ; 手动模式
LD W361.10  ; 进料伺服X轴#2夹爪配对取放料位触发标志
AND D1043.00  ; 进料伺服机构单步/自动循环运行中（总）
ORLD
AND=SL(303) D6166 D6004  ; 进料伺服X轴#2夹爪配对取放料位SV, 进料伺服X轴目标位置
ORLD
ANDLD
OUT 480.00  ; 进料伺服X轴定位目标位置设定OK

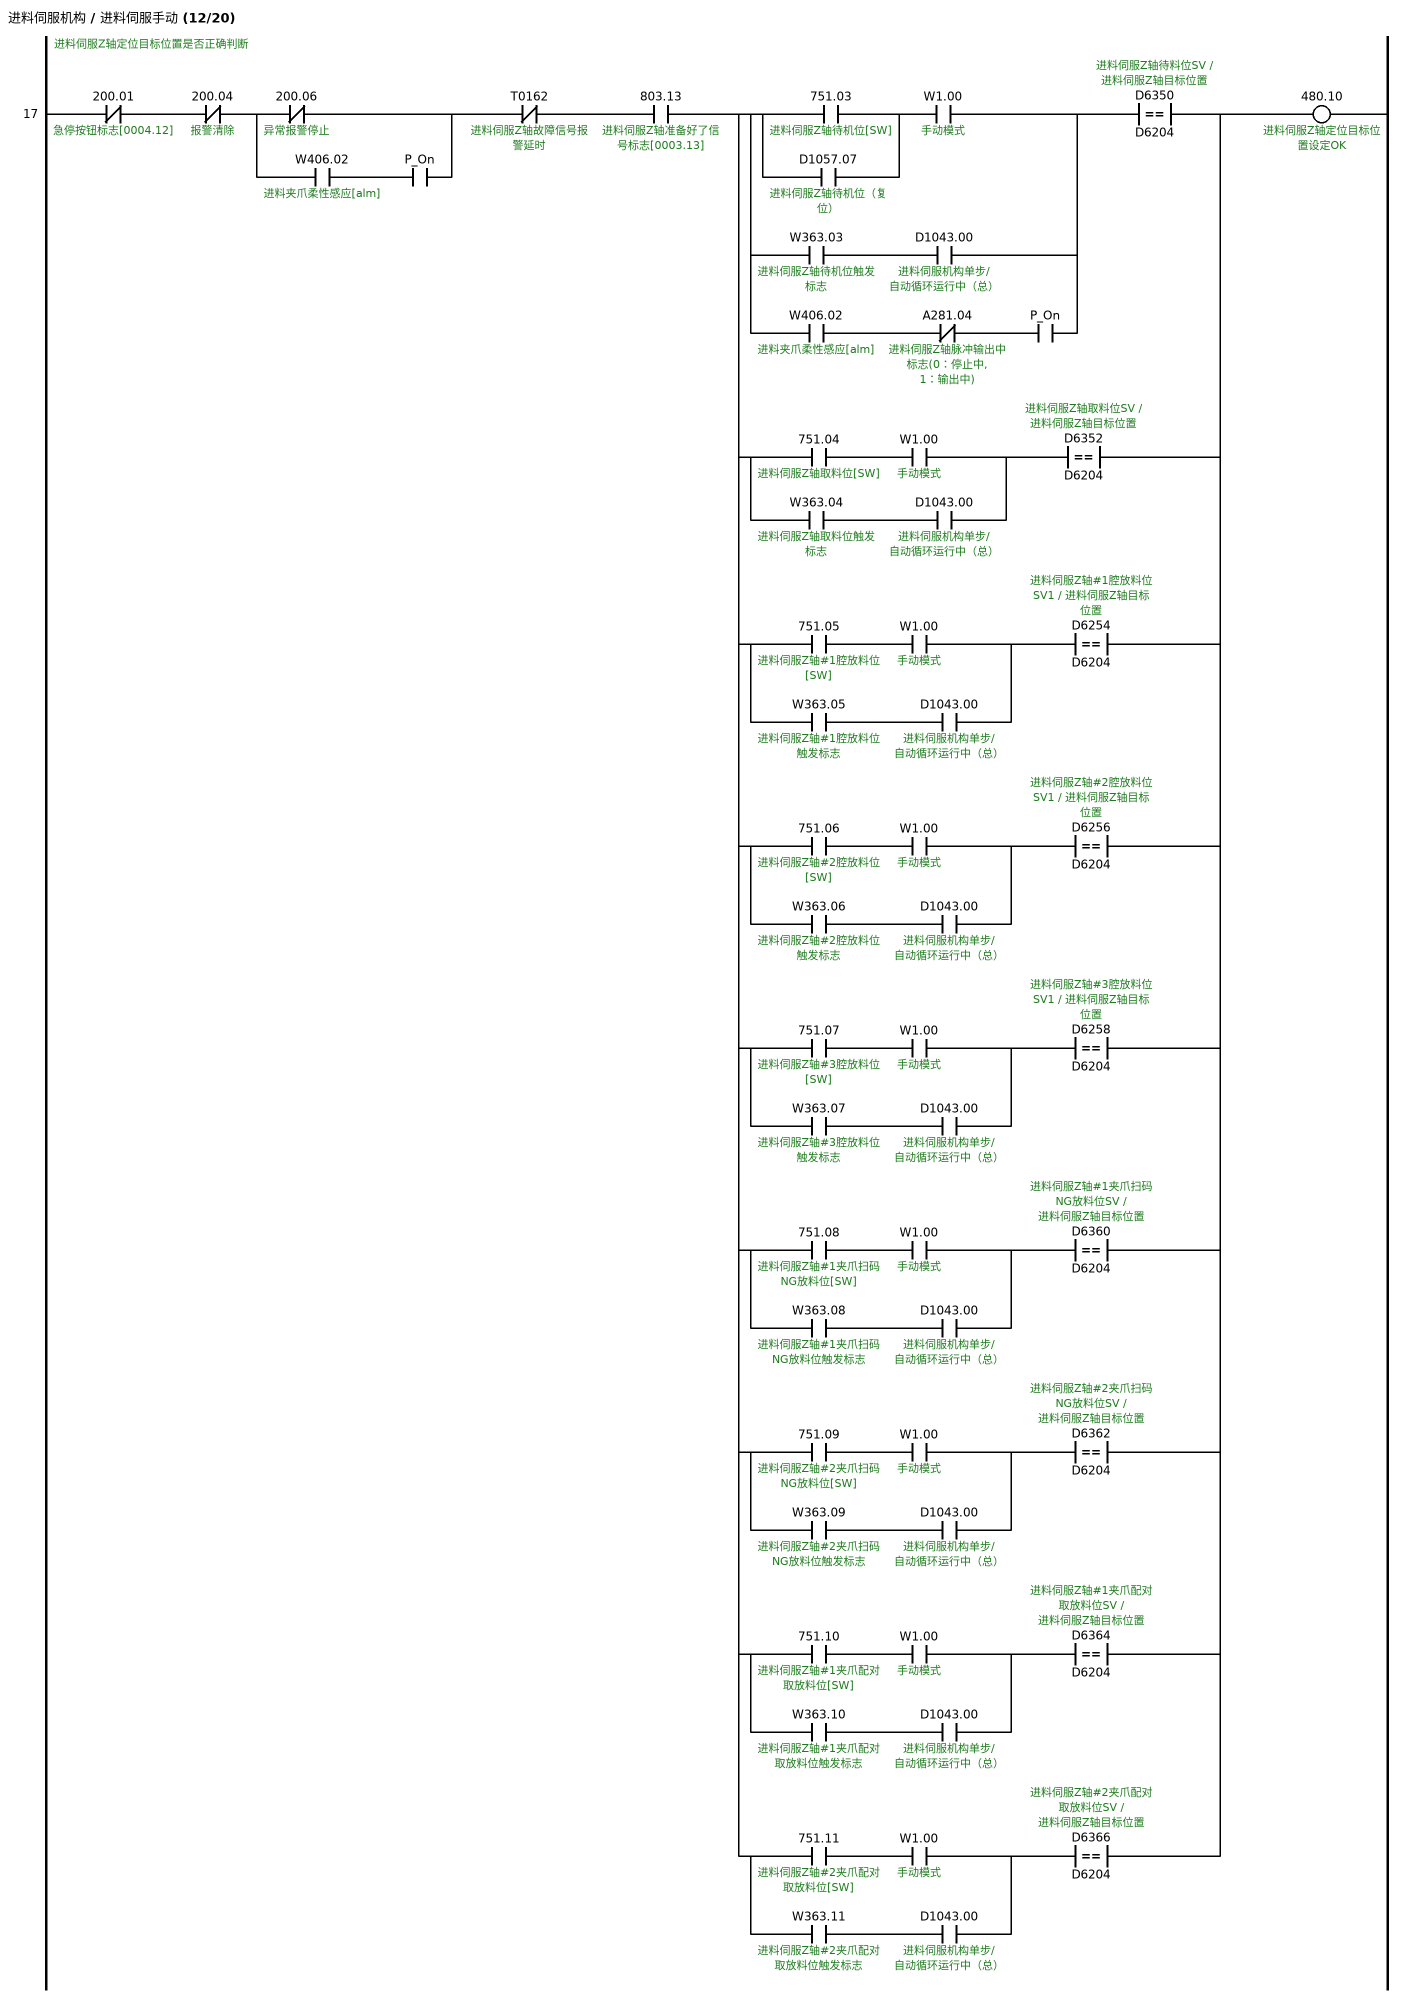
; rung 17: 进料伺服Z轴定位目标位置是否正确判断
LDNOT 200.01  ; 急停按钮标志[0004.12]
ANDNOT 200.04  ; 报警清除
LDNOT 200.06  ; 异常报警停止
LD W406.02  ; 进料夹爪柔性感应[alm]
AND P_On
ORLD
ANDLD
ANDNOT T0162  ; 进料伺服Z轴故障信号报警延时
AND 803.13  ; 进料伺服Z轴准备好了信号标志[0003.13]
LD 751.03  ; 进料伺服Z轴待机位[SW]
OR D1057.07  ; 进料伺服Z轴待机位（复位）
AND W1.00  ; 手动模式
LD W363.03  ; 进料伺服Z轴待机位触发标志
AND D1043.00  ; 进料伺服机构单步/自动循环运行中（总）
ORLD
LD W406.02  ; 进料夹爪柔性感应[alm]
ANDNOT A281.04  ; 进料伺服Z轴脉冲输出中标志(0：停止中,1：输出中)
AND P_On
ORLD
AND=SL(303) D6350 D6204  ; 进料伺服Z轴待料位SV, 进料伺服Z轴目标位置
LD 751.04  ; 进料伺服Z轴取料位[SW]
AND W1.00  ; 手动模式
LD W363.04  ; 进料伺服Z轴取料位触发标志
AND D1043.00  ; 进料伺服机构单步/自动循环运行中（总）
ORLD
AND=SL(303) D6352 D6204  ; 进料伺服Z轴取料位SV, 进料伺服Z轴目标位置
ORLD
LD 751.05  ; 进料伺服Z轴#1腔放料位[SW]
AND W1.00  ; 手动模式
LD W363.05  ; 进料伺服Z轴#1腔放料位触发标志
AND D1043.00  ; 进料伺服机构单步/自动循环运行中（总）
ORLD
AND=SL(303) D6254 D6204  ; 进料伺服Z轴#1腔放料位SV1, 进料伺服Z轴目标位置
ORLD
LD 751.06  ; 进料伺服Z轴#2腔放料位[SW]
AND W1.00  ; 手动模式
LD W363.06  ; 进料伺服Z轴#2腔放料位触发标志
AND D1043.00  ; 进料伺服机构单步/自动循环运行中（总）
ORLD
AND=SL(303) D6256 D6204  ; 进料伺服Z轴#2腔放料位SV1, 进料伺服Z轴目标位置
ORLD
LD 751.07  ; 进料伺服Z轴#3腔放料位[SW]
AND W1.00  ; 手动模式
LD W363.07  ; 进料伺服Z轴#3腔放料位触发标志
AND D1043.00  ; 进料伺服机构单步/自动循环运行中（总）
ORLD
AND=SL(303) D6258 D6204  ; 进料伺服Z轴#3腔放料位SV1, 进料伺服Z轴目标位置
ORLD
LD 751.08  ; 进料伺服Z轴#1夹爪扫码NG放料位[SW]
AND W1.00  ; 手动模式
LD W363.08  ; 进料伺服Z轴#1夹爪扫码NG放料位触发标志
AND D1043.00  ; 进料伺服机构单步/自动循环运行中（总）
ORLD
AND=SL(303) D6360 D6204  ; 进料伺服Z轴#1夹爪扫码NG放料位SV, 进料伺服Z轴目标位置
ORLD
LD 751.09  ; 进料伺服Z轴#2夹爪扫码NG放料位[SW]
AND W1.00  ; 手动模式
LD W363.09  ; 进料伺服Z轴#2夹爪扫码NG放料位触发标志
AND D1043.00  ; 进料伺服机构单步/自动循环运行中（总）
ORLD
AND=SL(303) D6362 D6204  ; 进料伺服Z轴#2夹爪扫码NG放料位SV, 进料伺服Z轴目标位置
ORLD
LD 751.10  ; 进料伺服Z轴#1夹爪配对取放料位[SW]
AND W1.00  ; 手动模式
LD W363.10  ; 进料伺服Z轴#1夹爪配对取放料位触发标志
AND D1043.00  ; 进料伺服机构单步/自动循环运行中（总）
ORLD
AND=SL(303) D6364 D6204  ; 进料伺服Z轴#1夹爪配对取放料位SV, 进料伺服Z轴目标位置
ORLD
LD 751.11  ; 进料伺服Z轴#2夹爪配对取放料位[SW]
AND W1.00  ; 手动模式
LD W363.11  ; 进料伺服Z轴#2夹爪配对取放料位触发标志
AND D1043.00  ; 进料伺服机构单步/自动循环运行中（总）
ORLD
AND=SL(303) D6366 D6204  ; 进料伺服Z轴#2夹爪配对取放料位SV, 进料伺服Z轴目标位置
ORLD
ANDLD
OUT 480.10  ; 进料伺服Z轴定位目标位置设定OK

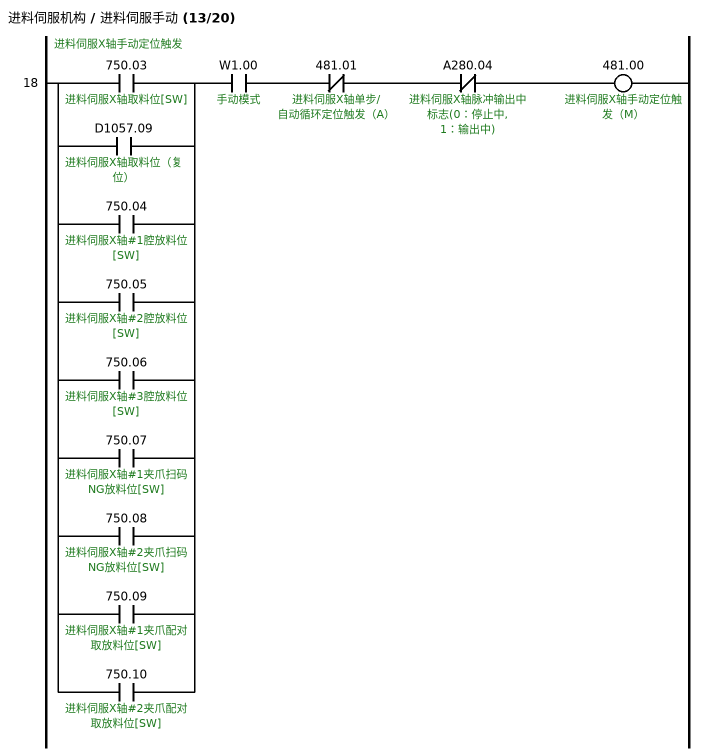
; rung 18: 进料伺服X轴手动定位触发
LD 750.03  ; 进料伺服X轴取料位[SW]
OR D1057.09  ; 进料伺服X轴取料位（复位）
OR 750.04  ; 进料伺服X轴#1腔放料位[SW]
OR 750.05  ; 进料伺服X轴#2腔放料位[SW]
OR 750.06  ; 进料伺服X轴#3腔放料位[SW]
OR 750.07  ; 进料伺服X轴#1夹爪扫码NG放料位[SW]
OR 750.08  ; 进料伺服X轴#2夹爪扫码NG放料位[SW]
OR 750.09  ; 进料伺服X轴#1夹爪配对取放料位[SW]
OR 750.10  ; 进料伺服X轴#2夹爪配对取放料位[SW]
AND W1.00  ; 手动模式
ANDNOT 481.01  ; 进料伺服X轴单步/自动循环定位触发（A）
ANDNOT A280.04  ; 进料伺服X轴脉冲输出中标志(0：停止中,1：输出中)
OUT 481.00  ; 进料伺服X轴手动定位触发（M）

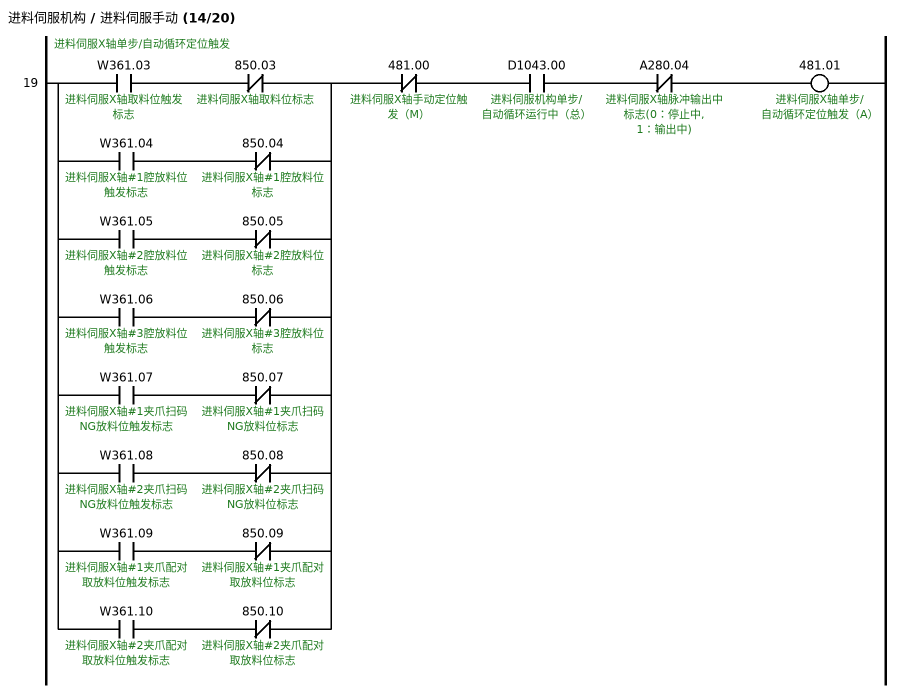
; rung 19: 进料伺服X轴单步/自动循环定位触发
LD W361.03  ; 进料伺服X轴取料位触发标志
ANDNOT 850.03  ; 进料伺服X轴取料位标志
LD W361.04  ; 进料伺服X轴#1腔放料位触发标志
ANDNOT 850.04  ; 进料伺服X轴#1腔放料位标志
ORLD
LD W361.05  ; 进料伺服X轴#2腔放料位触发标志
ANDNOT 850.05  ; 进料伺服X轴#2腔放料位标志
ORLD
LD W361.06  ; 进料伺服X轴#3腔放料位触发标志
ANDNOT 850.06  ; 进料伺服X轴#3腔放料位标志
ORLD
LD W361.07  ; 进料伺服X轴#1夹爪扫码NG放料位触发标志
ANDNOT 850.07  ; 进料伺服X轴#1夹爪扫码NG放料位标志
ORLD
LD W361.08  ; 进料伺服X轴#2夹爪扫码NG放料位触发标志
ANDNOT 850.08  ; 进料伺服X轴#2夹爪扫码NG放料位标志
ORLD
LD W361.09  ; 进料伺服X轴#1夹爪配对取放料位触发标志
ANDNOT 850.09  ; 进料伺服X轴#1夹爪配对取放料位标志
ORLD
LD W361.10  ; 进料伺服X轴#2夹爪配对取放料位触发标志
ANDNOT 850.10  ; 进料伺服X轴#2夹爪配对取放料位标志
ORLD
ANDNOT 481.00  ; 进料伺服X轴手动定位触发（M）
AND D1043.00  ; 进料伺服机构单步/自动循环运行中（总）
ANDNOT A280.04  ; 进料伺服X轴脉冲输出中标志(0：停止中,1：输出中)
OUT 481.01  ; 进料伺服X轴单步/自动循环定位触发（A）

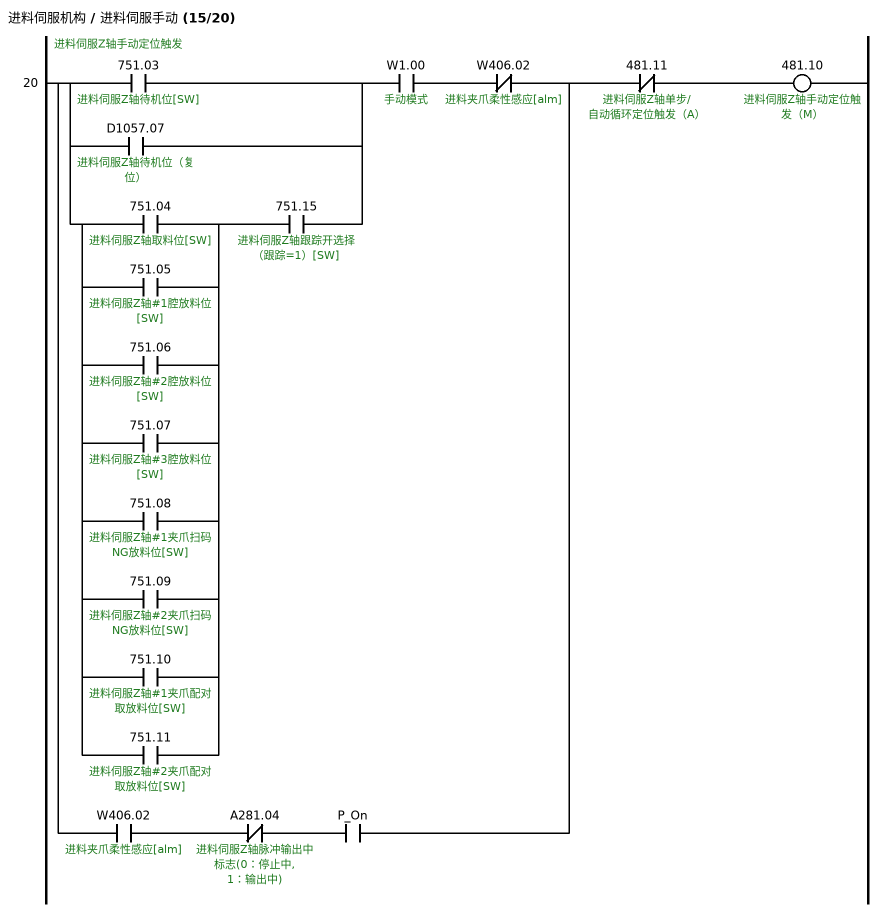
; rung 20: 进料伺服Z轴手动定位触发
LD 751.03  ; 进料伺服Z轴待机位[SW]
OR D1057.07  ; 进料伺服Z轴待机位（复位）
LD 751.04  ; 进料伺服Z轴取料位[SW]
OR 751.05  ; 进料伺服Z轴#1腔放料位[SW]
OR 751.06  ; 进料伺服Z轴#2腔放料位[SW]
OR 751.07  ; 进料伺服Z轴#3腔放料位[SW]
OR 751.08  ; 进料伺服Z轴#1夹爪扫码NG放料位[SW]
OR 751.09  ; 进料伺服Z轴#2夹爪扫码NG放料位[SW]
OR 751.10  ; 进料伺服Z轴#1夹爪配对取放料位[SW]
OR 751.11  ; 进料伺服Z轴#2夹爪配对取放料位[SW]
AND 751.15  ; 进料伺服Z轴跟踪开选择（跟踪=1）[SW]
ORLD
AND W1.00  ; 手动模式
ANDNOT W406.02  ; 进料夹爪柔性感应[alm]
LD W406.02  ; 进料夹爪柔性感应[alm]
ANDNOT A281.04  ; 进料伺服Z轴脉冲输出中标志(0：停止中,1：输出中)
AND P_On
ORLD
ANDNOT 481.11  ; 进料伺服Z轴单步/自动循环定位触发（A）
OUT 481.10  ; 进料伺服Z轴手动定位触发（M）

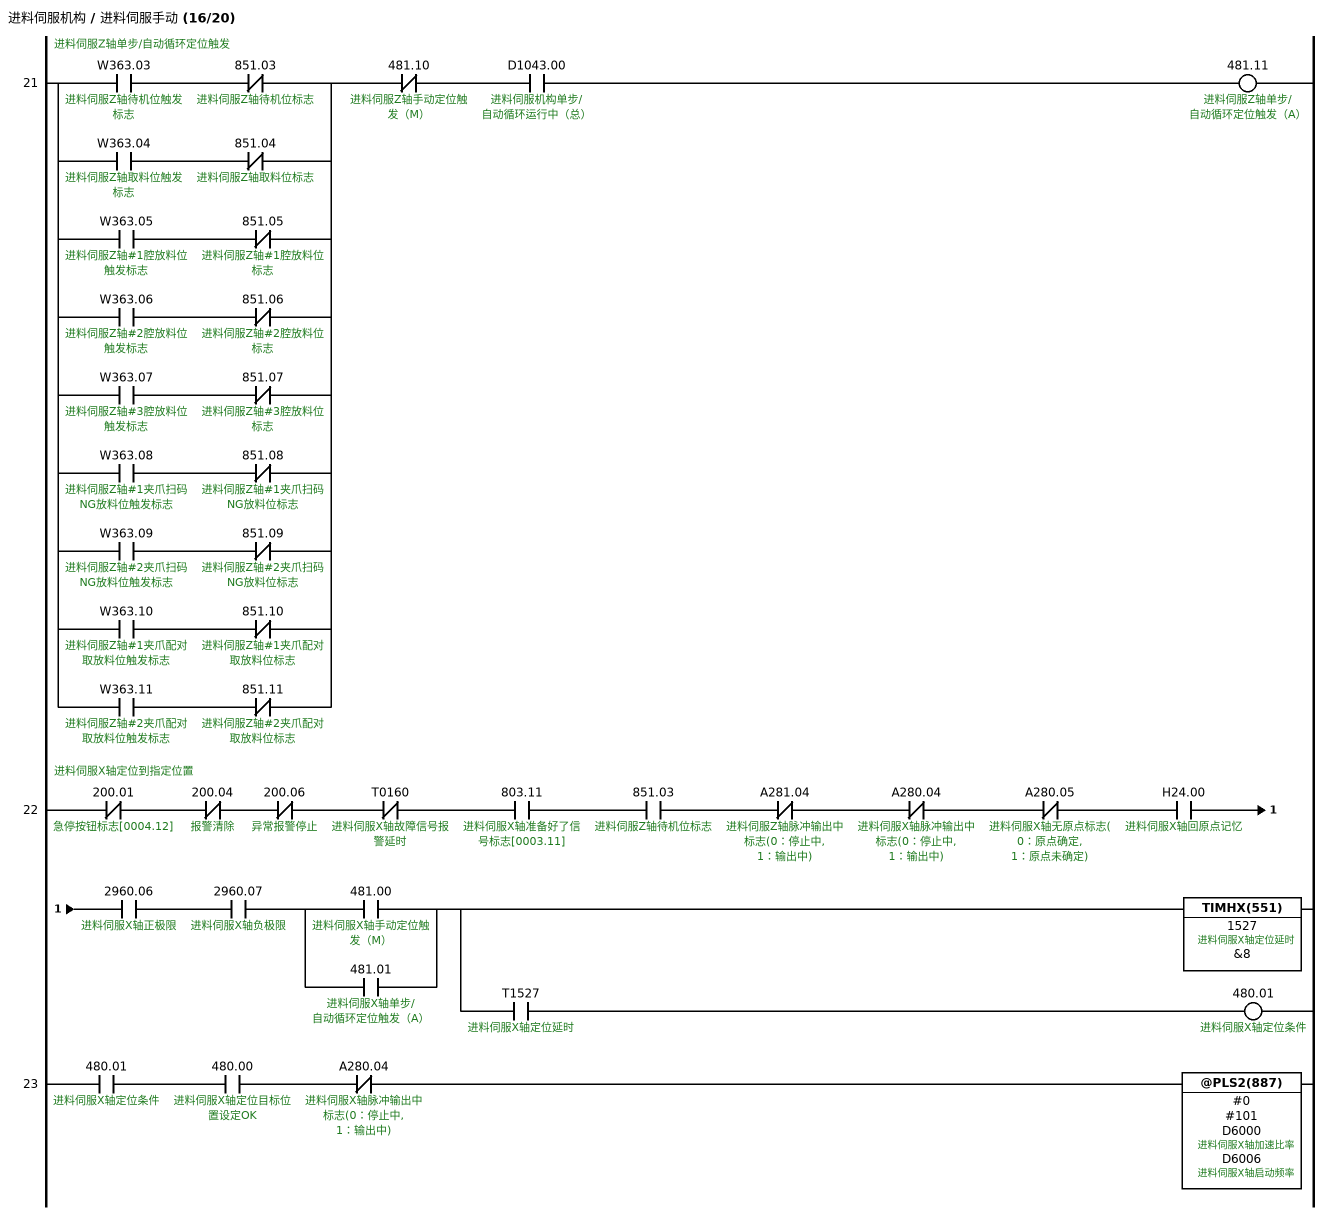
; rung 21: 进料伺服Z轴单步/自动循环定位触发
LD W363.03  ; 进料伺服Z轴待机位触发标志
ANDNOT 851.03  ; 进料伺服Z轴待机位标志
LD W363.04  ; 进料伺服Z轴取料位触发标志
ANDNOT 851.04  ; 进料伺服Z轴取料位标志
ORLD
LD W363.05  ; 进料伺服Z轴#1腔放料位触发标志
ANDNOT 851.05  ; 进料伺服Z轴#1腔放料位标志
ORLD
LD W363.06  ; 进料伺服Z轴#2腔放料位触发标志
ANDNOT 851.06  ; 进料伺服Z轴#2腔放料位标志
ORLD
LD W363.07  ; 进料伺服Z轴#3腔放料位触发标志
ANDNOT 851.07  ; 进料伺服Z轴#3腔放料位标志
ORLD
LD W363.08  ; 进料伺服Z轴#1夹爪扫码NG放料位触发标志
ANDNOT 851.08  ; 进料伺服Z轴#1夹爪扫码NG放料位标志
ORLD
LD W363.09  ; 进料伺服Z轴#2夹爪扫码NG放料位触发标志
ANDNOT 851.09  ; 进料伺服Z轴#2夹爪扫码NG放料位标志
ORLD
LD W363.10  ; 进料伺服Z轴#1夹爪配对取放料位触发标志
ANDNOT 851.10  ; 进料伺服Z轴#1夹爪配对取放料位标志
ORLD
LD W363.11  ; 进料伺服Z轴#2夹爪配对取放料位触发标志
ANDNOT 851.11  ; 进料伺服Z轴#2夹爪配对取放料位标志
ORLD
ANDNOT 481.10  ; 进料伺服Z轴手动定位触发（M）
AND D1043.00  ; 进料伺服机构单步/自动循环运行中（总）
OUT 481.11  ; 进料伺服Z轴单步/自动循环定位触发（A）
; rung 22: 进料伺服X轴定位到指定位置
LDNOT 200.01  ; 急停按钮标志[0004.12]
ANDNOT 200.04  ; 报警清除
ANDNOT 200.06  ; 异常报警停止
ANDNOT T0160  ; 进料伺服X轴故障信号报警延时
AND 803.11  ; 进料伺服X轴准备好了信号标志[0003.11]
AND 851.03  ; 进料伺服Z轴待机位标志
ANDNOT A281.04  ; 进料伺服Z轴脉冲输出中标志(0：停止中,1：输出中)
ANDNOT A280.04  ; 进料伺服X轴脉冲输出中标志(0：停止中,1：输出中)
ANDNOT A280.05  ; 进料伺服X轴无原点标志(0：原点确定,1：原点未确定)
AND H24.00  ; 进料伺服X轴回原点记忆
AND 2960.06  ; 进料伺服X轴正极限
AND 2960.07  ; 进料伺服X轴负极限
LD 481.00  ; 进料伺服X轴手动定位触发（M）
OR 481.01  ; 进料伺服X轴单步/自动循环定位触发（A）
ANDLD
TIMHX(551) 1527 &8  ; 进料伺服X轴定位延时
AND T1527  ; 进料伺服X轴定位延时
OUT 480.01  ; 进料伺服X轴定位条件
; rung 23
LD 480.01  ; 进料伺服X轴定位条件
AND 480.00  ; 进料伺服X轴定位目标位置设定OK
ANDNOT A280.04  ; 进料伺服X轴脉冲输出中标志(0：停止中,1：输出中)
@PLS2(887) #0 #101 D6000 D6006  ; 进料伺服X轴加速比率, 进料伺服X轴启动频率

